(* IEC 61131-3 sources: std_i2980_v2.06_cp053/Source/IMM/ieccontrol/AutoCalibration1 (part 3) *)

(* ---- ABAutoIdentSpeed.pu ---- *)
IMPORT_OVER_LISTFILE
 GET_SYNC_REFTO
, SET_ALARM
, SET_EVENT
, CHECK_REF
, cCompEjector
, cCompMold
, KSYS_Status_OK
, cOptionHydraulic
, tnCalibState_None
, tnCalibState_Running
, tnCalibCommand_Stop
, tnCalibState_Aborted
, cMoveFwd
, cMoveNone
, cMoveBwd
, cMoveDecompAftPlast
, tnCalibState_Error
, cCalibMovements
, nSetup
, tnCalibCommand_None
, tnCalibState_Done
, tnCalibCommand_Start
, tsGlobalIdentSpeedStatus
, tsIdentSpeedMovement
, tnOperationMode
, tyPumpData
, tevRedoIdentSpeedEvent
, tevStopRequest
, tevStartRequest
, tsDeviceId
, tpIdentSpeedMovement
, FBCheckReady
, tevStartRequestData
, tevStopRequestData
, FBIdentSpeedWriteLog
, ABAutoIdentSpeedMeasure
, tnDataState
, KSYS_Status
, tOptionId
, FBTracePendingAlarms
, tevRedoIdentSpeedEventData
, tsVelPre
, tyIdentSpeedMovements
, TON

END_IMPORT

ALGORITHM_BLOCK ABAutoIdentSpeed #DUMMY_EDIT_BLOCK

SYSTEM_VAR
 sv_GlobalIdentMaxSpeedStatus : tsGlobalIdentSpeedStatus;
 sv_EjectorIdentMaxMovement : tsIdentSpeedMovement;
 sv_MoldIdentMaxMovement : tsIdentSpeedMovement;
 sv_InjectionIdentMaxMovement : tsIdentSpeedMovement;
 sv_NozzleIdentMaxMovement : tsIdentSpeedMovement;
 sv_GlobalIdentMinSpeedStatus : tsGlobalIdentSpeedStatus;
 sv_EjectorIdentMinMovement : tsIdentSpeedMovement;
 sv_MoldIdentMinMovement : tsIdentSpeedMovement;
 sv_InjectionIdentMinMovement : tsIdentSpeedMovement;
 sv_NozzleIdentMinMovement : tsIdentSpeedMovement;
 sv_iPendingAlarms : DINT;
 sv_OperationMode : tnOperationMode;
 sv_bAutoIdentRunning : BOOL (* auto calibration active *);
 sv_bCoresActive : BOOL;
 sv_PumpData : tyPumpData;
 sv_DataState : tnDataState;
END_VAR

SYSTEM_OBJECT
 TaskMid : TASK;
 TaskSlow : TASK;
 TaskInject : TASK;
 TaskAnalog : TASK;
 PU_Task_7 : TASK;
 EV_Task_7 : TASK;
 erCalibrationSpeedStopped : ALARM;
 erSetupModeRequiredForCalib : ALARM;
 erCalibCoresActive : ALARM;
 evRedoIdentMaxSpeedStart : tevRedoIdentSpeedEvent;
 evRedoIdentMinSpeedStart : tevRedoIdentSpeedEvent;
 evStopRequest : tevStopRequest;
 evStartRequest : tevStartRequest;
 PU_Task_13 : TASK;
END_OBJECT

VAR
 DeviceIdEjector : tsDeviceId := (CompId:=cCompEjector,IndexId:=1);
 DeviceIdMold : tsDeviceId := (CompId:=cCompMold,IndexId:=1);
 mActMovement : tpIdentSpeedMovement;
 mCalibCounter : DINT;
 mbUseSingleMovement : BOOL;
 fbCheckReady : FBCheckReady;
 evStartRequestData : tevStartRequestData;
 evStopRequestData : tevStopRequestData;
 fbIdentWriteLog : FBIdentSpeedWriteLog;
 miFileCounter : UDINT;
 mbDeleteFiles : BOOL;
 mbLogFileSaved : BOOL := TRUE;
 msFileName : STRING(255);
 mbRestartMeas : BOOL;
 abSpeedMeasure : ABAutoIdentSpeedMeasure;
 mrRefVelocity : REAL;
 mrRefPressure : REAL;
 mrMaxLimitPosition : REAL;
 mrMinLimitPosition : REAL;
 dummy : DINT;
 mrMinPositionFactor : REAL := 0.2 (* 20% of stroke *);
 mrMaxPositionFactor : REAL := 0.8 (* 80% of stroke *);
 mrMaxVelocity : REAL;
 mrMaxPressure : REAL;
 mbVelocityLimitReached : BOOL;
 mbPressureLimitReached : BOOL;
 miErrorNo : INT;
 cIdentSpeedMaxSequence : INT := 100;
 cIdentSpeedMinSequence : INT := 200;
 cIdentSpeedMaxFwdIdent : INT := 101;
 cIdentSpeedMinFwdIdent : INT := 201;
 cIdentSpeedMaxBwdIdent : INT := 102;
 cIdentSpeedMinBwdIdent : INT := 202;
 cIdentSpeedMaxBwdInit : INT := 103;
 cIdentSpeedMinBwdInit : INT := 203;
 cIdentSpeedMaxFwdInit : INT := 104;
 cIdentSpeedMinFwdInit : INT := 204;
 cIdentSpeedMaxFwdStart : INT := 105;
 cIdentSpeedMinFwdStart : INT := 205;
 cIdentSpeedMaxBwdStart : INT := 106;
 cIdentSpeedMinBwdStart : INT := 206;
 cIdentSpeedMaxEnd : INT := 107;
 cIdentSpeedMinEnd : INT := 207;
 mrBwdStopPosition : REAL := 0.05;
 mprActPressure : REFTO REAL;
 mbprActPressureLinked : BOOL;
END_VAR

PROCESS_ALGORITHM paInit ON TaskMid AUTOSTART

VAR_TEMP
 j : DINT;
 k : DINT;
END_VAR

VAR
 i : DINT;
 Status : KSYS_Status;
 rpPosition : REFTO REAL;
 tmpM : tpIdentSpeedMovement;
 pOption : REFTO tOptionId;
END_VAR
#BEGIN_EDIT_BLOCK
(**************************************** WARNING ********************************************
 *** The KEBA Kemro K2 System including software is not intended for safety control tasks! ***
 ***                       For further information see Comment tab!                        ***
 *********************************************************************************************)

i := 1;

rpPosition := GET_SYNC_REFTO('Ejector1.ai_Position', T#0s, Status);
IF Status = KSYS_Status_OK THEN
    sv_GlobalIdentMaxSpeedStatus.pMovements[i] := @sv_EjectorIdentMaxMovement;
    sv_GlobalIdentMinSpeedStatus.pMovements[i] := @sv_EjectorIdentMinMovement;
    i := i + 1;
END_IF;

sv_GlobalIdentMaxSpeedStatus.pMovements[i] := @sv_MoldIdentMaxMovement;
sv_GlobalIdentMinSpeedStatus.pMovements[i] := @sv_MoldIdentMinMovement;
i := i + 1;

pOption := GET_SYNC_REFTO('Nozzle1.sv_Options', T#0s, Status);
IF (Status = KSYS_Status_OK) AND ((pOption^ AND cOptionHydraulic) = cOptionHydraulic) THEN;
    //hydraulic nozzle -> check if ai_Position is available
    rpPosition := GET_SYNC_REFTO('Nozzle1.ai_Position', T#0s, Status);
    IF Status = KSYS_Status_OK THEN
        sv_GlobalIdentMaxSpeedStatus.pMovements[i] := @sv_NozzleIdentMaxMovement;
        sv_GlobalIdentMinSpeedStatus.pMovements[i] := @sv_NozzleIdentMinMovement;
        i := i + 1;
    END_IF;
END_IF;

sv_GlobalIdentMaxSpeedStatus.pMovements[i] := @sv_InjectionIdentMaxMovement;
sv_GlobalIdentMinSpeedStatus.pMovements[i] := @sv_InjectionIdentMinMovement;
i := i + 1;

(* sort them by iOrder *)
FOR k := 1 TO i - 2 DO
    FOR j := 1 TO i - 1 - k DO
        IF sv_GlobalIdentMaxSpeedStatus.pMovements[j]^.iOrder > sv_GlobalIdentMaxSpeedStatus.pMovements[j + 1]^.iOrder THEN
            tmpM := sv_GlobalIdentMaxSpeedStatus.pMovements[j];
            sv_GlobalIdentMaxSpeedStatus.pMovements[j] := sv_GlobalIdentMaxSpeedStatus.pMovements[j + 1];
            sv_GlobalIdentMaxSpeedStatus.pMovements[j + 1] := tmpM;
            tmpM := sv_GlobalIdentMinSpeedStatus.pMovements[j];
            sv_GlobalIdentMinSpeedStatus.pMovements[j] := sv_GlobalIdentMinSpeedStatus.pMovements[j + 1];
            sv_GlobalIdentMinSpeedStatus.pMovements[j + 1] := tmpM;
        END_IF;
    END_FOR;
END_FOR;

sv_GlobalIdentMaxSpeedStatus.iMaxStep := i - 1;
sv_GlobalIdentMinSpeedStatus.iMaxStep := i - 1;

sv_GlobalIdentMaxSpeedStatus.iCurrentStep := 0;
sv_GlobalIdentMaxSpeedStatus.Status := tnCalibState_None;
sv_GlobalIdentMaxSpeedStatus.bInitDone := TRUE;

sv_GlobalIdentMinSpeedStatus.iCurrentStep := 0;
sv_GlobalIdentMinSpeedStatus.Status := tnCalibState_None;
sv_GlobalIdentMinSpeedStatus.bInitDone := TRUE;

STOP_PROCESS_ALGORITHM();

;#END_EDIT_BLOCK END_ALGORITHM

POSTUPDATE_ALGORITHM pAlarmPending ON PU_Task_7 WITH sv_iPendingAlarms

VAR
 fbTracePendingAlarms : FBTracePendingAlarms;
END_VAR
#BEGIN_EDIT_BLOCK
IF ((sv_GlobalIdentMaxSpeedStatus.Status = tnCalibState_Running) OR (sv_GlobalIdentMinSpeedStatus.Status = tnCalibState_Running)) AND
    (sv_iPendingAlarms <> 0) THEN

   dummy := Print('auto max. speed identification stopped because alarms of class 1/2/3 pending');

   //trace all pending alarms
   fbTracePendingAlarms();

   IF (sv_GlobalIdentMaxSpeedStatus.Status = tnCalibState_Running) THEN
      sv_GlobalIdentMaxSpeedStatus.Command := tnCalibCommand_Stop;
      sv_GlobalIdentMaxSpeedStatus.Status := tnCalibState_Aborted;
   ELSE
      sv_GlobalIdentMinSpeedStatus.Command := tnCalibCommand_Stop;
      sv_GlobalIdentMinSpeedStatus.Status := tnCalibState_Aborted;
   END_IF;

   SET_ALARM(Name := erCalibrationSpeedStopped,
             Param1 := miErrorNo);
END_IF;

;#END_EDIT_BLOCK END_ALGORITHM

ALGORITHM aMeasure

VAR
 rActPressure : REAL;
END_VAR
#BEGIN_EDIT_BLOCK
IF mbprActPressureLinked THEN
   rActPressure := mprActPressure^;
ELSE
   rActPressure := 0.0;
END_IF;
abSpeedMeasure.aMeasure(bRestart := mbRestartMeas,
                        rPosition := mActMovement^.prPosition^,
                        rRefVelocity := mrRefVelocity,
                        rActVelocity := mActMovement^.prActVelocity^,
                        rRefPressure := mrRefPressure,
                        rActPressure := rActPressure,
                        rMaxLimitPosition := mrMaxLimitPosition,
                        rMinLimitPosition := mrMinLimitPosition);
mbRestartMeas := FALSE;

;#END_EDIT_BLOCK END_ALGORITHM

PROCESS_ALGORITHM paMeasureFast ON TaskInject

#BEGIN_EDIT_BLOCK
aMeasure();

;#END_EDIT_BLOCK END_ALGORITHM

PROCESS_ALGORITHM paMeasureMid ON TaskAnalog

#BEGIN_EDIT_BLOCK
aMeasure();

;#END_EDIT_BLOCK END_ALGORITHM

ALGORITHM aStartMeasurement

#BEGIN_EDIT_BLOCK
mbRestartMeas := TRUE;
abSpeedMeasure.aReset();
abSpeedMeasure.aMeasure(bRestart := TRUE);
START_PROCESS_ALGORITHM(paMeasureMid);

;#END_EDIT_BLOCK END_ALGORITHM

ALGORITHM aStopMeasurement

#BEGIN_EDIT_BLOCK
STOP_PROCESS_ALGORITHM(paMeasureMid);
abSpeedMeasure.aCloseMeasure();

;#END_EDIT_BLOCK END_ALGORITHM

ALGORITHM aWriteLog

VAR_INPUT
 sFileName : STRING(255) (* file name movement *);
 iFileCounter : UDINT (* actual ident cycle index *);
 bDeleteFiles : BOOL (* delete old files *);
END_VAR
#BEGIN_EDIT_BLOCK
mbLogFileSaved := FALSE;
msFileName := sFileName;
miFileCounter := iFileCounter;
mbDeleteFiles := bDeleteFiles;

START_PROCESS_ALGORITHM(paWriteLog);

;#END_EDIT_BLOCK END_ALGORITHM

PROCESS_ALGORITHM paWriteLog ON TaskSlow

#BEGIN_EDIT_BLOCK
fbIdentWriteLog(sFileName    := msFileName,
                iFileCounter := miFileCounter,
                bDeleteFiles := mbDeleteFiles,
                rMaxVelocity := mrMaxVelocity,
                rMaxPressure := mrMaxPressure,
                bVelocityLimitReached := mbVelocityLimitReached,
                bPressureLimitReached := mbPressureLimitReached);
IF fbIdentWriteLog.bDone THEN
   mbLogFileSaved := TRUE;
ELSE
   mbLogFileSaved := FALSE;
END_IF;
STOP_PROCESS_ALGORITHM();

;#END_EDIT_BLOCK END_ALGORITHM

ALGORITHM aStartMovementFwd

#BEGIN_EDIT_BLOCK
IF mActMovement^.bPositionIncreasingFwd THEN
   mActMovement^.prIdentPosition^ := mActMovement^.prStroke^ * mrMaxPositionFactor;
ELSE
   mActMovement^.prIdentPosition^ := mActMovement^.prStroke^ * mrMinPositionFactor;
END_IF;
mActMovement^.pbMoveIdent^ := TRUE;

evStartRequestData.DeviceId := mActMovement^.DeviceId;
evStartRequestData.MoveDir := cMoveFwd;
IF mActMovement^.MoveId > cMoveNone THEN
   evStartRequestData.MoveId := mActMovement^.MoveId;
ELSE
   evStartRequestData.MoveId := cMoveFwd;
END_IF;

SET_EVENT(evStartRequest, evStartRequestData);

;#END_EDIT_BLOCK END_ALGORITHM

ALGORITHM aStartMovementBwd

#BEGIN_EDIT_BLOCK
IF mActMovement^.bPositionIncreasingFwd THEN
   mActMovement^.prIdentPosition^ := mActMovement^.prStroke^ * mrMinPositionFactor;
ELSE
   mActMovement^.prIdentPosition^ := mActMovement^.prStroke^ * mrMaxPositionFactor;
END_IF;
mActMovement^.pbMoveIdent^ := TRUE;

evStartRequestData.DeviceId := mActMovement^.DeviceId;
evStartRequestData.MoveDir := cMoveBwd;
IF mActMovement^.MoveId > cMoveNone THEN
   evStartRequestData.MoveId := cMoveDecompAftPlast;
ELSE
   evStartRequestData.MoveId := cMoveBwd;
END_IF;

SET_EVENT(evStartRequest, evStartRequestData);

;#END_EDIT_BLOCK END_ALGORITHM

ALGORITHM aStopMovementFwd

#BEGIN_EDIT_BLOCK
evStopRequestData.DeviceId := mActMovement^.DeviceId;
evStopRequestData.MoveDir := cMoveFwd;
evStopRequestData.MoveId := cMoveFwd;
SET_EVENT(evStopRequest, evStopRequestData);
mActMovement^.pbMoveIdent^ := FALSE;
mActMovement^.prIdentPosition^ := 0.0;
mActMovement^.prStopRamp^ := 0.0;

;#END_EDIT_BLOCK END_ALGORITHM

ALGORITHM aStopMovementBwd

#BEGIN_EDIT_BLOCK
evStopRequestData.DeviceId := mActMovement^.DeviceId;
evStopRequestData.MoveDir := cMoveBwd;
IF mActMovement^.MoveId > cMoveNone THEN
   evStopRequestData.MoveId := cMoveDecompAftPlast;
ELSE
   evStopRequestData.MoveId := cMoveBwd;
END_IF;
SET_EVENT(evStopRequest, evStopRequestData);
mActMovement^.pbMoveIdent^ := FALSE;
mActMovement^.prIdentPosition^ := 0.0;
mActMovement^.prStopRamp^ := 0.0;

;#END_EDIT_BLOCK END_ALGORITHM

ALGORITHM aStopMovementError

VAR_INPUT
 sMovementName : STRING(255) (* Movement information *);
END_VAR
#BEGIN_EDIT_BLOCK
sv_GlobalIdentMinSpeedStatus.Status := tnCalibState_Aborted;
mActMovement^.Status := tnCalibState_Error;

dummy := Print('Calib movement "%s" aborted.', sMovementName);

;#END_EDIT_BLOCK END_ALGORITHM

ALGORITHM aCalcMaxSpeedOutput

VAR_INPUT
 rMaxSpeedLimit : REAL (* Maximum speed limit of actual device *);
 rActSpeedLimit : REAL (* Actual speed limit of actual device *);
 rActMaxSpeed : REAL (* Maximum measured speed *);
 bPresLimitReached : BOOL (* Pressure limit reached during movement *);
 bUsePressureMode : BOOL (* Use pressure to check maimum speed limit reached. Otherwise use actual  velocity *);
END_VAR

VAR_OUTPUT
 bMaxDetected : BOOL (* Speed limit detected *);
 rRefSpeed : REAL (* Speed limit for next try *);
 rMaxSpeed : REAL (* Identified max speed *);
END_VAR

VAR
 rSpeedReachedFactor : REAL := 0.95;
 rMaxActSpeed : REAL;
 rMinActSpeed : REAL := 0.0;
 rMinSpeedDifference : REAL := 0.05;
END_VAR
#BEGIN_EDIT_BLOCK
IF (bUsePressureMode) THEN
   IF (rMaxActSpeed = 0.0) THEN
      rMaxActSpeed := rMaxSpeedLimit;
   END_IF;
   IF (bPresLimitReached) THEN
      // reduce refernce value
      rMaxActSpeed := rActSpeedLimit;
      IF (ABS(rMaxActSpeed - rMinActSpeed) < rMinSpeedDifference * rMaxSpeedLimit) THEN
         bMaxDetected := TRUE;
         rMaxSpeed := rMinActSpeed;
         rMinActSpeed := 0.0;
         rMaxActSpeed := 0.0;
      ELSE
         bMaxDetected := FALSE;
         rRefSpeed := 0.5 * (rMaxActSpeed + rMinActSpeed);
      END_IF;
   ELSE
      // ccompare with old value
      IF (rActSpeedLimit = rMaxSpeedLimit) THEN // maximum used at start
         // maximum with tolerance reached
         bMaxDetected := TRUE;
         rMaxSpeed := rMaxSpeedLimit;
         rMinActSpeed := 0.0;
         rMaxActSpeed := 0.0;
      ELSE
         // increase
         rMinActSpeed := rActSpeedLimit;
         IF (ABS(rMaxActSpeed - rMinActSpeed) < rMinSpeedDifference * rMaxSpeedLimit) THEN
            bMaxDetected := TRUE;
            rMaxSpeed := rMinActSpeed;
            rMinActSpeed := 0.0;
            rMaxActSpeed := 0.0;
         ELSE
            rRefSpeed := 0.5 * (rMaxActSpeed + rMinActSpeed);
         END_IF;
      END_IF;
   END_IF;
ELSE
   IF (rActSpeedLimit = rMaxSpeedLimit) THEN // maximum used at start
      IF (rActMaxSpeed > rSpeedReachedFactor * rActSpeedLimit)  THEN
      // maximum with tolerance reached
         bMaxDetected := TRUE;
         rMaxSpeed := rMaxSpeedLimit;
      ELSE
      // actual speed lower than maximum with tolerance
         bMaxDetected := FALSE;
         rRefSpeed := rActMaxSpeed;
         rMaxActSpeed := rActMaxSpeed;
      END_IF;
   ELSE
      IF (rActMaxSpeed > rSpeedReachedFactor * rActSpeedLimit) THEN
      // reference speed with tolerance reached
         bMaxDetected := TRUE;
         rMaxSpeed := rRefSpeed;
      ELSE
      // actual speed lower than reference speed with tolerance reached
      // check calibration of pump/valve
         bMaxDetected := TRUE;
         rMaxSpeed := rRefSpeed;
      END_IF;
   END_IF;
END_IF;

;#END_EDIT_BLOCK END_ALGORITHM

EVENT_ALGORITHM evaRedoMaxEvent ON EV_Task_7 WITH evRedoIdentMaxSpeedStart

VAR_INPUT
 evRedoIdentEventData : tevRedoIdentSpeedEventData (* Event data to start max speed identification *);
END_VAR
#BEGIN_EDIT_BLOCK

START_PROCESS_ALGORITHM(paRedoMax);

;#END_EDIT_BLOCK END_ALGORITHM

PROCESS_ALGORITHM paRedoMax ON TaskMid

VAR_TEMP
 i : DINT;
 bIdentActive : BOOL;
END_VAR
#BEGIN_EDIT_BLOCK
bIdentActive := FALSE;
FOR i:= 1 TO cCalibMovements DO
   IF CHECK_REF(sv_GlobalIdentMaxSpeedStatus.pMovements[i]^) THEN
      IF sv_GlobalIdentMaxSpeedStatus.pMovements[i]^.bRedo THEN
         mActMovement := sv_GlobalIdentMaxSpeedStatus.pMovements[i];
         bIdentActive := TRUE;
         sv_GlobalIdentMaxSpeedStatus.iCurrentStep :=  i;
         mCalibCounter := i;
         IF sv_OperationMode = nSetup THEN
            mbUseSingleMovement := TRUE;
            START_PROCESS_ALGORITHM(paMaxSingleMovement);
         ELSE
            sv_GlobalIdentMaxSpeedStatus.pMovements[i]^.bRedo := FALSE;
            SET_ALARM(erSetupModeRequiredForCalib);
         END_IF;
         EXIT;
      END_IF;
   END_IF;
END_FOR;
IF ((NOT bIdentActive) AND (sv_GlobalIdentMaxSpeedStatus.Status = tnCalibState_Running)) THEN
   sv_GlobalIdentMaxSpeedStatus.Status := tnCalibState_Aborted;
END_IF;

STOP_PROCESS_ALGORITHM();

;#END_EDIT_BLOCK END_ALGORITHM

PROCESS_ALGORITHM paMaxSingleMovement ON TaskMid

VAR
 bMoveBwdDone : BOOL := FALSE;
 bMoveFwdDone : BOOL := FALSE;
 bMoveIdentDone : BOOL := FALSE;
 sFileName : STRING(255);
 iFileCounter : UDINT := 1;
 ConstVis : tsVelPre (* const output for ejector forward movement *);
 ConstVisFwd : tsVelPre (* const output for ejector forward movement *);
 ConstVisBwd : tsVelPre (* const output for ejector forward movement *);
 bMaxFwdRetry : BOOL;
 bMaxBwdRetry : BOOL;
 bMaxFwdDetected : BOOL;
 bMaxBwdDetected : BOOL;
 sMoveName : STRING(32);
 rMaxPressureLimit : REAL;
 rRefSpeedLimit : REAL;
 rSpeedLimitFwd : REAL;
 rSpeedLimitBwd : REAL;
 rMaxRefPressureLimit : REAL;
 sWriteSpeedLimit : STRING(255);
 rVelocitSizeFactor : REAL := 1.0;
 rStartFactor : REAL := 0.1;
 rMinStopRamp : REAL := 1.0;
 rMinStrokeFactor : REAL := 0.5;
 bDelayTimeOffFwdLinked : BOOL;
 bDelayTimeOffBwdLinked : BOOL;
 dDelayTimeOffFwd : TIME;
 dDelayTimeOffBwd : TIME;
 dMinDelayTimeOff : TIME := T#25ms;
END_VAR

(* IecGraph-Code *)

(* init step *)
INITIAL_STEP S_INIT:
Action3 (P);
END_STEP

ACTION Action3: #BEGIN_EDIT_BLOCK
miErrorNo := 0;

ConstVisFwd := mActMovement^.pConstFwdVis^;
ConstVisBwd := mActMovement^.pConstBwdVis^;

sv_GlobalIdentMaxSpeedStatus.Status := tnCalibState_Running;
mActMovement^.Status := tnCalibState_Running;
sMoveName := mActMovement^.sName;

abSpeedMeasure.aInit();

bMaxFwdRetry := FALSE;
bMaxBwdRetry := FALSE;

IF (mActMovement^.rMaxPositionLimitFactor > mActMovement^.rMinPositionLimitFactor) AND
   (mActMovement^.rMinPositionLimitFactor > 0.0) AND (mActMovement^.rMaxPositionLimitFactor < 1.0) THEN
   mrMaxPositionFactor := mActMovement^.rMaxPositionLimitFactor;
   mrMinPositionFactor := mActMovement^.rMinPositionLimitFactor;
ELSE // use deafult values
   mrMaxPositionFactor := 0.8;
   mrMinPositionFactor := 0.2;
END_IF;

mprActPressure := sv_PumpData[mActMovement^.DeviceId.IndexId].prActSysPressure;
IF CHECK_REF(mprActPressure^) THEN
   mbprActPressureLinked := TRUE;
ELSE
   mbprActPressureLinked := FALSE;
END_IF;

IF CHECK_REF(mActMovement^.pdDelayTimeOffFwd^) THEN
   bDelayTimeOffFwdLinked := TRUE;
   dDelayTimeOffFwd := mActMovement^.pdDelayTimeOffFwd^;
ELSE
   bDelayTimeOffFwdLinked := FALSE;
END_IF;
IF CHECK_REF(mActMovement^.pdDelayTimeOffBwd^) THEN
   bDelayTimeOffBwdLinked := TRUE;
   dDelayTimeOffBwd := mActMovement^.pdDelayTimeOffBwd^;
ELSE
   bDelayTimeOffBwdLinked := FALSE;
END_IF;

;#END_EDIT_BLOCK END_ACTION (*Action3*)

(* steps *)
STEP S_RESET:
END_STEP

STEP S_STOP:
AStopSelf (P);
END_STEP

ACTION AStopSelf: #BEGIN_EDIT_BLOCK
sv_GlobalIdentMaxSpeedStatus.Command := tnCalibCommand_None;
sv_bAutoIdentRunning := FALSE;
mActMovement^.bRedo := FALSE;
mActMovement^.prStopRamp^ := 0.0;
mActMovement^.pConstFwdVis^ := ConstVisFwd;
mActMovement^.pConstBwdVis^ := ConstVisBwd;

//release memory
abSpeedMeasure.aEnd();

STOP_PROCESS_ALGORITHM();

;#END_EDIT_BLOCK END_ACTION (*AStopSelf*)
STEP S_MoveStartBwd:
AMoveStartBwd (P);
ACheckMoveStartBwdReady (N);
AMoveStartBwdReady (P0);
END_STEP

ACTION AMoveStartBwd: #BEGIN_EDIT_BLOCK
bMoveBwdDone := FALSE;
miErrorNo := cIdentSpeedMaxBwdInit;
aStartMovementBwd();

;#END_EDIT_BLOCK END_ACTION (*AMoveStartBwd*)
ACTION ACheckMoveStartBwdReady: #BEGIN_EDIT_BLOCK
fbCheckReady(DeviceId := evStartRequestData.DeviceId);
IF fbCheckReady.bReady THEN
   bMoveBwdDone := TRUE;
END_IF;

;#END_EDIT_BLOCK END_ACTION (*ACheckMoveStartBwdReady*)
ACTION AMoveStartBwdReady: #BEGIN_EDIT_BLOCK
aStopMovementBwd();

;#END_EDIT_BLOCK END_ACTION (*AMoveStartBwdReady*)
STEP S_StopMoveStartBwd:
AStopMoveStartBwd (P);
END_STEP

ACTION AStopMoveStartBwd: #BEGIN_EDIT_BLOCK
aStopMovementError(sMovementName := CONCAT(sMoveName, ' max ident Fwd: Bwd to initial position'));

;#END_EDIT_BLOCK END_ACTION (*AStopMoveStartBwd*)
STEP S_CHECK_ALARMS_INITBWD:
END_STEP

STEP S_INITCALIB_FWD:
aInitIdentFwd (P);
END_STEP

ACTION aInitIdentFwd: #BEGIN_EDIT_BLOCK
iFileCounter := 1;
IF (CHECK_REF(mActMovement^.prSizeFactorFwd^)) THEN
   IF (mActMovement^.prSizeFactorFwd^ > 0.0) THEN
      rVelocitSizeFactor := mActMovement^.prSizeFactorFwd^;
   END_IF;
ELSE
   rVelocitSizeFactor := 1.0;
END_IF;
rRefSpeedLimit := mActMovement^.prVelocityLimitFwd^;
rMaxPressureLimit := mActMovement^.prMaxPressureFwd^;
IF CHECK_REF(mActMovement^.prMaxPressureFwdHydr^) THEN
   rMaxRefPressureLimit := mActMovement^.prMaxPressureFwdHydr^;
ELSE
   rMaxRefPressureLimit := rMaxPressureLimit;
END_IF;

dummy := Print('Calib max speed %s Fwd started', sMoveName);

;#END_EDIT_BLOCK END_ACTION (*aInitIdentFwd*)
STEP S_CALIB_FWD:
ADoCalib (P);
AStartMovementFwd (P);
ACheckActMovementFwdReady (N);
AStopMovementFwd (P0);
END_STEP

ACTION ADoCalib: #BEGIN_EDIT_BLOCK
(* start calibration *)
// save actual settings
ConstVis := mActMovement^.pConstFwdVis^;

mActMovement^.pConstFwdVis^.Velocity.Output.rOutputValue := rRefSpeedLimit * rVelocitSizeFactor;
mActMovement^.pConstFwdVis^.Velocity.rMinOutput := 0.0;
mActMovement^.pConstFwdVis^.Pressure.Output.rOutputValue := MAX(mActMovement^.pConstFwdVis^.Pressure.Output.rOutputValue, rMaxPressureLimit);
mActMovement^.pConstFwdVis^.Pressure.Output.rRamp := MAX(1.0e9,ConstVis.Pressure.Output.rRamp);
IF mActMovement^.bPositionIncreasingFwd THEN
   mActMovement^.prIdentPosition^ := mActMovement^.prStroke^ * mrMaxPositionFactor;
   mrMinLimitPosition := rStartFactor * mActMovement^.prIdentPosition^ + (1.0 - rStartFactor) * mActMovement^.prPosition^;
   IF (mActMovement^.prIdentPosition^ - mActMovement^.prPosition^) > 0.0 THEN
      rMinStopRamp := rMinStrokeFactor * rRefSpeedLimit  * rRefSpeedLimit/ ABS(mActMovement^.prIdentPosition^ - mActMovement^.prPosition^);
   ELSE
      rMinStopRamp := 0.0;
   END_IF;
   mActMovement^.prStopRamp^ := MAX(mActMovement^.pConstFwdVis^.Velocity.Output.rRamp, rMinStopRamp);
   mrMaxLimitPosition := mActMovement^.prIdentPosition^;
ELSE
   mActMovement^.prIdentPosition^ := mActMovement^.prStroke^ * mrMinPositionFactor;
   mrMaxLimitPosition := (1.0 - rStartFactor) * mActMovement^.prPosition^ + rStartFactor * mActMovement^.prIdentPosition^;
   IF (mActMovement^.prPosition^ - mActMovement^.prIdentPosition^) > 0.0 THEN
      rMinStopRamp := rMinStrokeFactor * rRefSpeedLimit * rRefSpeedLimit / ABS(mActMovement^.prIdentPosition^ - mActMovement^.prPosition^);
   ELSE
      rMinStopRamp := 0.0;
   END_IF;
   mActMovement^.prStopRamp^ := MAX(mActMovement^.pConstFwdVis^.Velocity.Output.rRamp, rMinStopRamp);
   mrMinLimitPosition := mActMovement^.prIdentPosition^;
END_IF;
mActMovement^.pbMoveIdent^ := TRUE;
bMoveIdentDone := FALSE;

bMaxFwdDetected := FALSE;

mrRefVelocity := rRefSpeedLimit;
mrRefPressure := rMaxRefPressureLimit;
mbRestartMeas := TRUE;

IF bDelayTimeOffFwdLinked THEN
   mActMovement^.pdDelayTimeOffFwd^ := MAX(mActMovement^.pdDelayTimeOffFwd^, dMinDelayTimeOff);
END_IF;
IF bDelayTimeOffBwdLinked THEN
   mActMovement^.pdDelayTimeOffBwd^ := MAX(mActMovement^.pdDelayTimeOffBwd^, dMinDelayTimeOff);
END_IF;

aStartMeasurement();

sWriteSpeedLimit := REAL_TO_STRING(rRefSpeedLimit);
dummy := Print('Calib max output: act. max speed: %s', sWriteSpeedLimit);
miErrorNo := cIdentSpeedMaxFwdIdent;

;#END_EDIT_BLOCK END_ACTION (*ADoCalib*)
ACTION AStartMovementFwd: #BEGIN_EDIT_BLOCK
evStartRequestData.DeviceId := mActMovement^.DeviceId;
evStartRequestData.MoveDir := cMoveFwd;
IF mActMovement^.MoveId > cMoveNone THEN
   evStartRequestData.MoveId := mActMovement^.MoveId;
ELSE
   evStartRequestData.MoveId := cMoveFwd;
END_IF;
SET_EVENT(evStartRequest, evStartRequestData);

;#END_EDIT_BLOCK END_ACTION (*AStartMovementFwd*)
ACTION ACheckActMovementFwdReady: #BEGIN_EDIT_BLOCK
fbCheckReady(DeviceId := evStartRequestData.DeviceId);
IF fbCheckReady.bReady THEN
   bMoveIdentDone := TRUE;
END_IF;

;#END_EDIT_BLOCK END_ACTION (*ACheckActMovementFwdReady*)
ACTION AStopMovementFwd: #BEGIN_EDIT_BLOCK
aStopMeasurement();
aStopMovementFwd();

mActMovement^.pConstFwdVis^ := ConstVis;
mActMovement^.prStopRamp^ := 0.0;

IF bDelayTimeOffFwdLinked THEN
   mActMovement^.pdDelayTimeOffFwd^ := dDelayTimeOffFwd;
END_IF;
IF bDelayTimeOffBwdLinked THEN
   mActMovement^.pdDelayTimeOffBwd^ := dDelayTimeOffBwd;
END_IF;

;#END_EDIT_BLOCK END_ACTION (*AStopMovementFwd*)
STEP S_StopIdentFwd:
AStopIdentFwd (P);
END_STEP

ACTION AStopIdentFwd: #BEGIN_EDIT_BLOCK
aStopMovementError(sMovementName := CONCAT(sMoveName, ' max ident Fwd'));

;#END_EDIT_BLOCK END_ACTION (*AStopIdentFwd*)
STEP S_CHECK_ALARMS_FWD:
END_STEP

STEP S_WRITE_FWD:
AWriteFwd (P);
END_STEP

ACTION AWriteFwd: #BEGIN_EDIT_BLOCK
abSpeedMeasure.aGetMaxValues(rMaxSpeed => mrMaxVelocity,
                             rMaxPressure => mrMaxPressure,
                             bPressureLimitReached => mbPressureLimitReached,
                             bSpeedLimitReached => mbVelocityLimitReached);
sFileName := CONCAT(sMoveName,"_MAXSPEED_FWD_");
aWriteLog(sFileName := sFileName,
          iFileCounter := iFileCounter,
          bDeleteFiles := TRUE);
iFileCounter := iFileCounter + 1;

;#END_EDIT_BLOCK END_ACTION (*AWriteFwd*)
STEP S_AbortedWriteFwd:
AAbortedWriteFwd (P);
END_STEP

ACTION AAbortedWriteFwd: #BEGIN_EDIT_BLOCK
mActMovement^.Status := tnCalibState_Error;

;#END_EDIT_BLOCK END_ACTION (*AAbortedWriteFwd*)
STEP S_CHECK_MAXSPEED_FWD:
ACheckMaxSpeedFwd (P);
END_STEP

ACTION ACheckMaxSpeedFwd: #BEGIN_EDIT_BLOCK
aCalcMaxSpeedOutput(rMaxSpeedLimit := mActMovement^.prVelocityLimitFwd^,
                    rActSpeedLimit := rRefSpeedLimit,
                    rActMaxSpeed := abSpeedMeasure.aGetMaxValues.rMaxSpeed,
                    bPresLimitReached := abSpeedMeasure.aGetMaxValues.bPressureLimitReached,
                    bUsePressureMode := (mrMaxPressure > 0.0));
bMaxFwdDetected := aCalcMaxSpeedOutput.bMaxDetected;
IF (bMaxFwdDetected) THEN
   rSpeedLimitFwd := rRefSpeedLimit;
   dummy := Print('Calib max output %s Fwd finished: max speed fwd = %f$N', sMoveName, rSpeedLimitFwd);
ELSE
   IF abSpeedMeasure.aGetMaxValues.bPressureLimitReached THEN
      sWriteSpeedLimit := REAL_TO_STRING(rRefSpeedLimit);
      dummy := Print('Calib max output: pressure limit reached with act. max speed %s', sWriteSpeedLimit);
   END_IF;
   bMaxFwdRetry := TRUE;
   rRefSpeedLimit := aCalcMaxSpeedOutput.rRefSpeed;
END_IF;

;#END_EDIT_BLOCK END_ACTION (*ACheckMaxSpeedFwd*)
STEP S_MaxFwdRetry:
AStartMovementFwdBwd (P);
ACheckActMovementFwdBwdReady (N);
AStopMovementFwdBwd (P0);
END_STEP

ACTION AStartMovementFwdBwd: #BEGIN_EDIT_BLOCK
bMoveBwdDone := FALSE;
miErrorNo := cIdentSpeedMaxFwdStart;
aStartMovementBwd();

;#END_EDIT_BLOCK END_ACTION (*AStartMovementFwdBwd*)
ACTION ACheckActMovementFwdBwdReady: #BEGIN_EDIT_BLOCK
fbCheckReady(DeviceId := evStartRequestData.DeviceId);
IF fbCheckReady.bReady THEN
   bMoveBwdDone := TRUE;
END_IF;

;#END_EDIT_BLOCK END_ACTION (*ACheckActMovementFwdBwdReady*)
ACTION AStopMovementFwdBwd: #BEGIN_EDIT_BLOCK
aStopMovementBwd();

;#END_EDIT_BLOCK END_ACTION (*AStopMovementFwdBwd*)
STEP S_StopMoveBwd:
AStopMoveBwd (P);
END_STEP

ACTION AStopMoveBwd: #BEGIN_EDIT_BLOCK
aStopMovementError(sMovementName := CONCAT(sMoveName, ' max ident Fwd: Bwd to start position'));

;#END_EDIT_BLOCK END_ACTION (*AStopMoveBwd*)
STEP S_CHECK_ALARMS_RETRYFWD:
END_STEP

STEP S_InitStartMovementBwdFwd:
AInitStartMovementBwdFwd (P);
ACheckInitMovementBwdFwdReady (N);
AStopInitMovementBwdFwd (P0);
END_STEP

ACTION AInitStartMovementBwdFwd: #BEGIN_EDIT_BLOCK
bMoveFwdDone := FALSE;
miErrorNo := cIdentSpeedMaxFwdInit;
aStartMovementFwd();

;#END_EDIT_BLOCK END_ACTION (*AInitStartMovementBwdFwd*)
ACTION ACheckInitMovementBwdFwdReady: #BEGIN_EDIT_BLOCK
fbCheckReady(DeviceId := evStartRequestData.DeviceId);
IF fbCheckReady.bReady THEN
   bMoveFwdDone := TRUE;
END_IF;

;#END_EDIT_BLOCK END_ACTION (*ACheckInitMovementBwdFwdReady*)
ACTION AStopInitMovementBwdFwd: #BEGIN_EDIT_BLOCK
aStopMovementFwd();

;#END_EDIT_BLOCK END_ACTION (*AStopInitMovementBwdFwd*)
STEP S_StopInitMoveFwd:
AStopInitMoveFwd (P);
END_STEP

ACTION AStopInitMoveFwd: #BEGIN_EDIT_BLOCK
aStopMovementError(sMovementName := CONCAT(sMoveName, ' max ident Bwd: Fwd to initial position'));

;#END_EDIT_BLOCK END_ACTION (*AStopInitMoveFwd*)
STEP S_CHECK_ALARMS_STARTBWD:
END_STEP

STEP S_INITCALIB_BWD:
AInitCalibBwd (P);
END_STEP

ACTION AInitCalibBwd: #BEGIN_EDIT_BLOCK
iFileCounter := 1;
IF (CHECK_REF(mActMovement^.prSizeFactorBwd^)) THEN
   IF (mActMovement^.prSizeFactorBwd^ > 0.0) THEN
      rVelocitSizeFactor := mActMovement^.prSizeFactorBwd^;
   END_IF;
ELSE
   rVelocitSizeFactor := 1.0;
END_IF;
rRefSpeedLimit := mActMovement^.prVelocityLimitBwd^;
rMaxPressureLimit := mActMovement^.prMaxPressureBwd^;
IF CHECK_REF(mActMovement^.prMaxPressureBwdHydr^) THEN
   rMaxRefPressureLimit := mActMovement^.prMaxPressureBwdHydr^;
ELSE
   rMaxRefPressureLimit := mActMovement^.prMaxPressureFwd^;
END_IF;

dummy := Print('Calib max speed %s Bwd started', sMoveName);

;#END_EDIT_BLOCK END_ACTION (*AInitCalibBwd*)
STEP S_CALIB_BWD:
ADoCalibBwd (P);
AStartMovementBwd (P);
ACheckActMovementBwdReady (N);
AStopMovementBwd (P0);
END_STEP

ACTION ADoCalibBwd: #BEGIN_EDIT_BLOCK
ConstVis := mActMovement^.pConstBwdVis^;

mActMovement^.pConstBwdVis^.Velocity.Output.rOutputValue := rRefSpeedLimit * rVelocitSizeFactor;
mActMovement^.pConstBwdVis^.Velocity.rMinOutput := 0.0;
mActMovement^.pConstBwdVis^.Pressure.Output.rOutputValue := MAX(mActMovement^.pConstBwdVis^.Pressure.Output.rOutputValue, rMaxPressureLimit);
mActMovement^.pConstBwdVis^.Pressure.Output.rRamp := MAX(1.0e9,ConstVis.Pressure.Output.rRamp);
IF mActMovement^.bPositionIncreasingFwd THEN
   mActMovement^.prIdentPosition^ := mActMovement^.prStroke^ * mrMinPositionFactor;
   mrMaxLimitPosition := rStartFactor * mActMovement^.prIdentPosition^ + (1.0 - rStartFactor) * mActMovement^.prPosition^;
   rMinStopRamp := rRefSpeedLimit / ABS(mActMovement^.prIdentPosition^ - mActMovement^.prPosition^);
   IF (mActMovement^.prPosition^ - mActMovement^.prIdentPosition^) > 0.0 THEN
      rMinStopRamp := rMinStrokeFactor * rRefSpeedLimit * rRefSpeedLimit / ABS(mActMovement^.prIdentPosition^ - mActMovement^.prPosition^);
   ELSE
      rMinStopRamp := 0.0;
   END_IF;
   mActMovement^.prStopRamp^ := MAX(mActMovement^.pConstBwdVis^.Velocity.Output.rRamp, rMinStopRamp);
   mrMinLimitPosition := mActMovement^.prIdentPosition^;
ELSE
   mActMovement^.prIdentPosition^ := mActMovement^.prStroke^ * mrMaxPositionFactor;
   mrMinLimitPosition := rStartFactor * mActMovement^.prPosition^ + (1.0 - rStartFactor) * mActMovement^.prIdentPosition^;
   IF (mActMovement^.prIdentPosition^ - mActMovement^.prPosition^) > 0.0 THEN
      rMinStopRamp := rMinStrokeFactor * rRefSpeedLimit * rRefSpeedLimit / ABS(mActMovement^.prIdentPosition^ - mActMovement^.prPosition^);
   ELSE
      rMinStopRamp := 0.0;
   END_IF;
   mActMovement^.prStopRamp^ := MAX(mActMovement^.pConstBwdVis^.Velocity.Output.rRamp, rMinStopRamp);
   mrMaxLimitPosition := mActMovement^.prIdentPosition^;
END_IF;
mActMovement^.pbMoveIdent^ := TRUE;

bMoveIdentDone := FALSE;

mrRefVelocity := rRefSpeedLimit;
mrRefPressure := rMaxRefPressureLimit;
mbRestartMeas := TRUE;

IF bDelayTimeOffFwdLinked THEN
   mActMovement^.pdDelayTimeOffFwd^ := MAX(mActMovement^.pdDelayTimeOffFwd^, dMinDelayTimeOff);
END_IF;
IF bDelayTimeOffBwdLinked THEN
   mActMovement^.pdDelayTimeOffBwd^ := MAX(mActMovement^.pdDelayTimeOffBwd^, dMinDelayTimeOff);
END_IF;

aStartMeasurement();

sWriteSpeedLimit := REAL_TO_STRING(rRefSpeedLimit);
dummy := Print('Calib max output: act. max speed: %s', sWriteSpeedLimit);
miErrorNo := cIdentSpeedMaxBwdIdent;

;#END_EDIT_BLOCK END_ACTION (*ADoCalibBwd*)
ACTION AStartMovementBwd: #BEGIN_EDIT_BLOCK
evStartRequestData.DeviceId := mActMovement^.DeviceId;
evStartRequestData.MoveDir := cMoveBwd;
IF mActMovement^.MoveId > cMoveNone THEN
   evStartRequestData.MoveId := cMoveDecompAftPlast;
ELSE
   evStartRequestData.MoveId := cMoveBwd;
END_IF;
SET_EVENT(evStartRequest, evStartRequestData);

;#END_EDIT_BLOCK END_ACTION (*AStartMovementBwd*)
ACTION ACheckActMovementBwdReady: #BEGIN_EDIT_BLOCK
fbCheckReady(DeviceId := evStartRequestData.DeviceId);
IF fbCheckReady.bReady THEN
   bMoveIdentDone := TRUE;
END_IF;

;#END_EDIT_BLOCK END_ACTION (*ACheckActMovementBwdReady*)
ACTION AStopMovementBwd: #BEGIN_EDIT_BLOCK
aStopMeasurement();
aStopMovementBwd();

mActMovement^.pConstBwdVis^ := ConstVis;
mActMovement^.prStopRamp^ := 0.0;

IF bDelayTimeOffFwdLinked THEN
   mActMovement^.pdDelayTimeOffFwd^ := dDelayTimeOffFwd;
END_IF;
IF bDelayTimeOffBwdLinked THEN
   mActMovement^.pdDelayTimeOffBwd^ := dDelayTimeOffBwd;
END_IF;

;#END_EDIT_BLOCK END_ACTION (*AStopMovementBwd*)
STEP S_StopCalibBwd:
AStopCalibBwd (P);
END_STEP

ACTION AStopCalibBwd: #BEGIN_EDIT_BLOCK
aStopMovementError(sMovementName := CONCAT(sMoveName, ' max ident Bwd'));

;#END_EDIT_BLOCK END_ACTION (*AStopCalibBwd*)
STEP S_CHECK_ALARMS_BWD:
END_STEP

STEP S_WRITE_BWD:
AWriteBwd (P);
END_STEP

ACTION AWriteBwd: #BEGIN_EDIT_BLOCK
abSpeedMeasure.aGetMaxValues(rMaxSpeed => mrMaxVelocity,
                             rMaxPressure => mrMaxPressure,
                             bPressureLimitReached => mbPressureLimitReached,
                             bSpeedLimitReached => mbVelocityLimitReached);
sFileName := CONCAT(sMoveName,"_MAXSPEED_BWD_");
aWriteLog(sFileName := sFileName,
          iFileCounter := iFileCounter,
          bDeleteFiles := TRUE);
iFileCounter := iFileCounter + 1;

;#END_EDIT_BLOCK END_ACTION (*AWriteBwd*)
STEP S_CHECK_MAXSPEED_BWD:
ACheckMaxSpeedBwd (P);
END_STEP

ACTION ACheckMaxSpeedBwd: #BEGIN_EDIT_BLOCK
aCalcMaxSpeedOutput(rMaxSpeedLimit := mActMovement^.prVelocityLimitBwd^,
                    rActSpeedLimit := rRefSpeedLimit,
                    rActMaxSpeed := abSpeedMeasure.aGetMaxValues.rMaxSpeed,
                    bPresLimitReached := abSpeedMeasure.aGetMaxValues.bPressureLimitReached,
                    bUsePressureMode := (mrMaxPressure > 0.0));
bMaxBwdDetected := aCalcMaxSpeedOutput.bMaxDetected;
IF (bMaxBwdDetected) THEN
   rSpeedLimitBwd := rRefSpeedLimit;
   dummy := Print('Calib max output %s Bwd finished: max speed bwd = %f$N', sMoveName, rSpeedLimitBwd);
ELSE
   IF abSpeedMeasure.aGetMaxValues.bPressureLimitReached THEN
      sWriteSpeedLimit := REAL_TO_STRING(rRefSpeedLimit);
      dummy := Print('Calib max output: pressure limit reached with act. max speed %s', sWriteSpeedLimit);
   END_IF;
   bMaxBwdRetry := TRUE;
   rRefSpeedLimit := aCalcMaxSpeedOutput.rRefSpeed;
END_IF;

;#END_EDIT_BLOCK END_ACTION (*ACheckMaxSpeedBwd*)
STEP S_MaxBwdRetry:
AStartMovementBwdFwd (P);
ACheckActMovementBwdFwdReady (N);
AStopMovementBwdFwd (P0);
END_STEP

ACTION AStartMovementBwdFwd: #BEGIN_EDIT_BLOCK
bMoveFwdDone := FALSE;
miErrorNo := cIdentSpeedMaxBwdStart;
aStartMovementFwd();

;#END_EDIT_BLOCK END_ACTION (*AStartMovementBwdFwd*)
ACTION ACheckActMovementBwdFwdReady: #BEGIN_EDIT_BLOCK
fbCheckReady(DeviceId := evStartRequestData.DeviceId);
IF fbCheckReady.bReady THEN
   bMoveFwdDone := TRUE;
END_IF;

;#END_EDIT_BLOCK END_ACTION (*ACheckActMovementBwdFwdReady*)
ACTION AStopMovementBwdFwd: #BEGIN_EDIT_BLOCK
aStopMovementFwd();

;#END_EDIT_BLOCK END_ACTION (*AStopMovementBwdFwd*)
STEP S_StopMoveFwd:
AStopMoveFwd (P);
END_STEP

ACTION AStopMoveFwd: #BEGIN_EDIT_BLOCK
aStopMovementError(sMovementName := CONCAT(sMoveName, ' max ident Bwd: Fwd to start position'));

;#END_EDIT_BLOCK END_ACTION (*AStopMoveFwd*)
STEP S_CHECK_ALARMS_RETRYBWD:
END_STEP

STEP S_MoveEndBwd:
AMoveEndBwd (P);
ACheckMoveEndBwdReady (N);
AMoveEndBwdReady (P0);
END_STEP

ACTION AMoveEndBwd: #BEGIN_EDIT_BLOCK
bMoveBwdDone := FALSE;

IF mActMovement^.bPositionIncreasingFwd THEN
   mActMovement^.prIdentPosition^ := mrBwdStopPosition;
ELSE
   mActMovement^.prIdentPosition^ := mActMovement^.prStroke^ - mrBwdStopPosition;
END_IF;
mActMovement^.prStopRamp^ := 1.0e10;
mActMovement^.pConstBwdVis^.Pressure.Output.rRamp := MAX(1.0e20,mActMovement^.pConstBwdVis^.Pressure.Output.rRamp);
mActMovement^.pConstBwdVis^.Pressure.rMinOutput := 0.1 * rMaxPressureLimit;
sv_EjectorIdentMinMovement.pConstBwdVis^.Pressure.Output.rRamp := MAX(1.0e10, sv_EjectorIdentMinMovement.pConstBwdVis^.Pressure.Output.rRamp);
sv_EjectorIdentMinMovement.pConstBwdVis^.Pressure.rMinOutput := 0.1 * sv_EjectorIdentMinMovement.prMaxPressureBwd^;

mActMovement^.pbMoveIdent^ := TRUE;

evStartRequestData.DeviceId := mActMovement^.DeviceId;
evStartRequestData.MoveDir := cMoveBwd;
IF mActMovement^.MoveId > cMoveNone THEN
   evStartRequestData.MoveId := cMoveDecompAftPlast;
ELSE
   evStartRequestData.MoveId := cMoveBwd;
END_IF;
miErrorNo := cIdentSpeedMaxEnd;

SET_EVENT(evStartRequest, evStartRequestData);

;#END_EDIT_BLOCK END_ACTION (*AMoveEndBwd*)
ACTION ACheckMoveEndBwdReady: #BEGIN_EDIT_BLOCK
fbCheckReady(DeviceId := evStartRequestData.DeviceId);
IF fbCheckReady.bReady THEN
   bMoveBwdDone := TRUE;
END_IF;

;#END_EDIT_BLOCK END_ACTION (*ACheckMoveEndBwdReady*)
ACTION AMoveEndBwdReady: #BEGIN_EDIT_BLOCK
aStopMovementBwd();

;#END_EDIT_BLOCK END_ACTION (*AMoveEndBwdReady*)
STEP S_StopMoveEndBwd:
AStopMoveEndBwd (P);
END_STEP

ACTION AStopMoveEndBwd: #BEGIN_EDIT_BLOCK
aStopMovementError(sMovementName := CONCAT(sMoveName, ' max ident Bwd to end position'));

;#END_EDIT_BLOCK END_ACTION (*AStopMoveEndBwd*)
STEP S_Done:
ADone (P);
END_STEP

ACTION ADone: #BEGIN_EDIT_BLOCK
mActMovement^.Status := tnCalibState_Done;
sv_GlobalIdentMaxSpeedStatus.Status := tnCalibState_Done;

mActMovement^.prVelocityFwd^ := rSpeedLimitFwd;
mActMovement^.prVelocityBwd^ := rSpeedLimitBwd;

;#END_EDIT_BLOCK END_ACTION (*ADone*)

(* transitions *)
TRANSITION Trans47 (* Trans47 *) FROM S_RESET TO S_STOP :=  #BEGIN_EDIT_BLOCK
mbLogFileSaved
;#END_EDIT_BLOCK
END_TRANSITION

TRANSITION TRestart (* TRestart *) FROM S_STOP TO S_INIT :=  #BEGIN_EDIT_BLOCK
TRUE
;#END_EDIT_BLOCK
END_TRANSITION

TRANSITION TMoveStartBwd (* TMoveStartBwd *) FROM S_INIT TO S_MoveStartBwd :=  #BEGIN_EDIT_BLOCK
TRUE

;#END_EDIT_BLOCK
END_TRANSITION

TRANSITION TInitBwd (* TInitBwd *) FROM S_MoveStartBwd TO S_CHECK_ALARMS_INITBWD :=  #BEGIN_EDIT_BLOCK
bMoveBwdDone
;#END_EDIT_BLOCK
END_TRANSITION

GO_ON_TRANSITION TStopMoveStartBwd (* TStopMoveStartBwd *) FROM S_MoveStartBwd TO S_StopMoveStartBwd :=  #BEGIN_EDIT_BLOCK
sv_GlobalIdentMaxSpeedStatus.Status = tnCalibState_Aborted OR
sv_GlobalIdentMaxSpeedStatus.Status = tnCalibState_None
OR sv_iPendingAlarms <> 0
OR mActMovement^.bRedo = FALSE
;#END_EDIT_BLOCK
END_TRANSITION

GO_ON_TRANSITION TReset (* TReset *) FROM S_StopMoveStartBwd TO S_RESET :=  #BEGIN_EDIT_BLOCK
TRUE
;#END_EDIT_BLOCK
END_TRANSITION

TRANSITION TStartIdent (* TStartIdent *) FROM S_CHECK_ALARMS_INITBWD TO S_INITCALIB_FWD :=  #BEGIN_EDIT_BLOCK
S_CHECK_ALARMS_INITBWD.T > T#100ms
;#END_EDIT_BLOCK
END_TRANSITION

GO_ON_TRANSITION TStopInitBwd (* TStopInitBwd *) FROM S_CHECK_ALARMS_INITBWD TO S_StopMoveStartBwd :=  #BEGIN_EDIT_BLOCK
sv_iPendingAlarms <> 0
;#END_EDIT_BLOCK
END_TRANSITION

TRANSITION TDelay1 (* TDelay1 *) FROM S_INITCALIB_FWD TO S_CALIB_FWD :=  #BEGIN_EDIT_BLOCK
S_INITCALIB_FWD.T>T#1s
;#END_EDIT_BLOCK
END_TRANSITION

TRANSITION TMoveIdentFwdDone (* TMoveIdentFwdDone *) FROM S_CALIB_FWD TO S_CHECK_ALARMS_FWD :=  #BEGIN_EDIT_BLOCK
bMoveIdentDone
;#END_EDIT_BLOCK
END_TRANSITION

GO_ON_TRANSITION TStopIdentFwd (* TStopIdentFwd *) FROM S_CALIB_FWD TO S_StopIdentFwd :=  #BEGIN_EDIT_BLOCK
sv_GlobalIdentMaxSpeedStatus.Status = tnCalibState_Aborted OR
sv_GlobalIdentMaxSpeedStatus.Status = tnCalibState_None
OR sv_iPendingAlarms <> 0
OR mActMovement^.bRedo = FALSE
;#END_EDIT_BLOCK
END_TRANSITION

GO_ON_TRANSITION TReset1 (* TReset1 *) FROM S_StopIdentFwd TO S_RESET :=  #BEGIN_EDIT_BLOCK
TRUE
;#END_EDIT_BLOCK
END_TRANSITION

TRANSITION TStartWriteFwd (* TStartWriteFwd *) FROM S_CHECK_ALARMS_FWD TO S_WRITE_FWD :=  #BEGIN_EDIT_BLOCK
S_CHECK_ALARMS_FWD.T > T#100ms
;#END_EDIT_BLOCK
END_TRANSITION

GO_ON_TRANSITION TStopIdentFwd2 (* TStopIdentFwd2 *) FROM S_CHECK_ALARMS_FWD TO S_StopIdentFwd :=  #BEGIN_EDIT_BLOCK
sv_iPendingAlarms <> 0
;#END_EDIT_BLOCK
END_TRANSITION

TRANSITION TWriteFwd (* TWriteFwd *) FROM S_WRITE_FWD TO S_CHECK_MAXSPEED_FWD :=  #BEGIN_EDIT_BLOCK
mbLogFileSaved
;#END_EDIT_BLOCK
END_TRANSITION

GO_ON_TRANSITION TAbortedWriteFwd (* TAbortedWriteFwd *) FROM S_WRITE_FWD TO S_AbortedWriteFwd :=  #BEGIN_EDIT_BLOCK
sv_GlobalIdentMaxSpeedStatus.Status = tnCalibState_Aborted
;#END_EDIT_BLOCK
END_TRANSITION

GO_ON_TRANSITION TResetAbortedWriteFwd (* TResetAbortedWriteFwd *) FROM S_AbortedWriteFwd TO S_RESET :=  #BEGIN_EDIT_BLOCK
TRUE
;#END_EDIT_BLOCK
END_TRANSITION

TRANSITION TMaxFwdDetected (* TMaxFwdDetected *) FROM S_CHECK_MAXSPEED_FWD TO S_InitStartMovementBwdFwd :=  #BEGIN_EDIT_BLOCK
bMaxFwdDetected
;#END_EDIT_BLOCK
END_TRANSITION

TRANSITION Trans15 (* Trans15 *) FROM S_CHECK_MAXSPEED_FWD TO S_MaxFwdRetry :=  #BEGIN_EDIT_BLOCK
bMaxFwdRetry
;#END_EDIT_BLOCK
END_TRANSITION

TRANSITION TMoveBwdDone (* TMoveBwdDone *) FROM S_MaxFwdRetry TO S_CHECK_ALARMS_RETRYFWD :=  #BEGIN_EDIT_BLOCK
bMoveBwdDone
;#END_EDIT_BLOCK
END_TRANSITION

GO_ON_TRANSITION TStopMoveBwd (* TStopMoveBwd *) FROM S_MaxFwdRetry TO S_StopMoveBwd :=  #BEGIN_EDIT_BLOCK
sv_GlobalIdentMaxSpeedStatus.Status = tnCalibState_Aborted OR
sv_GlobalIdentMaxSpeedStatus.Status = tnCalibState_None
OR sv_iPendingAlarms <> 0
OR mActMovement^.bRedo = FALSE

;#END_EDIT_BLOCK
END_TRANSITION

TRANSITION TReset2 (* TReset2 *) FROM S_StopMoveBwd TO S_RESET :=  #BEGIN_EDIT_BLOCK
TRUE
;#END_EDIT_BLOCK
END_TRANSITION

TRANSITION TRetryFwd (* TRetryFwd *) FROM S_CHECK_ALARMS_RETRYFWD TO S_CALIB_FWD :=  #BEGIN_EDIT_BLOCK
S_CHECK_ALARMS_RETRYFWD.T > T#1s
;#END_EDIT_BLOCK
END_TRANSITION

GO_ON_TRANSITION TStopIdentFwd4 (* TStopIdentFwd4 *) FROM S_CHECK_ALARMS_RETRYFWD TO S_StopMoveBwd :=  #BEGIN_EDIT_BLOCK
sv_iPendingAlarms <> 0
;#END_EDIT_BLOCK
END_TRANSITION

TRANSITION Trans35 (* Trans35 *) FROM S_InitStartMovementBwdFwd TO S_CHECK_ALARMS_STARTBWD :=  #BEGIN_EDIT_BLOCK
bMoveFwdDone
;#END_EDIT_BLOCK
END_TRANSITION

GO_ON_TRANSITION TStopInitMoveFwd (* TStopInitMoveFwd *) FROM S_InitStartMovementBwdFwd TO S_StopInitMoveFwd :=  #BEGIN_EDIT_BLOCK
sv_GlobalIdentMaxSpeedStatus.Status = tnCalibState_Aborted OR
sv_GlobalIdentMaxSpeedStatus.Status = tnCalibState_None
OR sv_iPendingAlarms <> 0
OR mActMovement^.bRedo = FALSE
;#END_EDIT_BLOCK
END_TRANSITION

TRANSITION TResetInitMoveFwd (* TResetInitMoveFwd *) FROM S_StopInitMoveFwd TO S_RESET :=  #BEGIN_EDIT_BLOCK
TRUE
;#END_EDIT_BLOCK
END_TRANSITION

TRANSITION TStartInitBwd (* TStartInitBwd *) FROM S_CHECK_ALARMS_STARTBWD TO S_INITCALIB_BWD :=  #BEGIN_EDIT_BLOCK
S_CHECK_ALARMS_STARTBWD.T > T#100ms
;#END_EDIT_BLOCK
END_TRANSITION

GO_ON_TRANSITION TStopIdentFwd3 (* TStopIdentFwd3 *) FROM S_CHECK_ALARMS_STARTBWD TO S_StopInitMoveFwd :=  #BEGIN_EDIT_BLOCK
sv_iPendingAlarms <> 0
;#END_EDIT_BLOCK
END_TRANSITION

TRANSITION TInitCalibBwd (* TInitCalibBwd *) FROM S_INITCALIB_BWD TO S_CALIB_BWD :=  #BEGIN_EDIT_BLOCK
S_INITCALIB_BWD.T>T#1s
;#END_EDIT_BLOCK
END_TRANSITION

TRANSITION Trans14 (* Trans14 *) FROM S_CALIB_BWD TO S_CHECK_ALARMS_BWD :=  #BEGIN_EDIT_BLOCK
bMoveIdentDone
;#END_EDIT_BLOCK
END_TRANSITION

GO_ON_TRANSITION TStopCalibBwd (* TStopCalibBwd *) FROM S_CALIB_BWD TO S_StopCalibBwd :=  #BEGIN_EDIT_BLOCK
sv_GlobalIdentMaxSpeedStatus.Status = tnCalibState_Aborted OR
sv_GlobalIdentMaxSpeedStatus.Status = tnCalibState_None
OR sv_iPendingAlarms <> 0
OR mActMovement^.bRedo = FALSE
;#END_EDIT_BLOCK
END_TRANSITION

GO_ON_TRANSITION TResetCalibBwd (* TResetCalibBwd *) FROM S_StopCalibBwd TO S_RESET :=  #BEGIN_EDIT_BLOCK
TRUE
;#END_EDIT_BLOCK
END_TRANSITION

TRANSITION TStartWriteBwd (* TStartWriteBwd *) FROM S_CHECK_ALARMS_BWD TO S_WRITE_BWD :=  #BEGIN_EDIT_BLOCK
S_CHECK_ALARMS_BWD.T > T#100ms
;#END_EDIT_BLOCK
END_TRANSITION

GO_ON_TRANSITION TStopCalibBwd2 (* TStopCalibBwd2 *) FROM S_CHECK_ALARMS_BWD TO S_StopCalibBwd :=  #BEGIN_EDIT_BLOCK
sv_iPendingAlarms <> 0
;#END_EDIT_BLOCK
END_TRANSITION

TRANSITION TWriteBwd (* TWriteBwd *) FROM S_WRITE_BWD TO S_CHECK_MAXSPEED_BWD :=  #BEGIN_EDIT_BLOCK
mbLogFileSaved
;#END_EDIT_BLOCK
END_TRANSITION

TRANSITION TMaxBwdDetected (* TMaxBwdDetected *) FROM S_CHECK_MAXSPEED_BWD TO S_MoveEndBwd :=  #BEGIN_EDIT_BLOCK
bMaxBwdDetected
;#END_EDIT_BLOCK
END_TRANSITION

TRANSITION TMaxBwdRetry (* TMaxBwdRetry *) FROM S_CHECK_MAXSPEED_BWD TO S_MaxBwdRetry :=  #BEGIN_EDIT_BLOCK
bMaxBwdRetry
;#END_EDIT_BLOCK
END_TRANSITION

TRANSITION TMoveFwdDone (* TMoveFwdDone *) FROM S_MaxBwdRetry TO S_CHECK_ALARMS_RETRYBWD :=  #BEGIN_EDIT_BLOCK
bMoveFwdDone
;#END_EDIT_BLOCK
END_TRANSITION

GO_ON_TRANSITION TStopMoveFwd (* TStopMoveFwd *) FROM S_MaxBwdRetry TO S_StopMoveFwd :=  #BEGIN_EDIT_BLOCK
sv_GlobalIdentMaxSpeedStatus.Status = tnCalibState_Aborted OR
sv_GlobalIdentMaxSpeedStatus.Status = tnCalibState_None
OR sv_iPendingAlarms <> 0
OR mActMovement^.bRedo = FALSE

;#END_EDIT_BLOCK
END_TRANSITION

TRANSITION TResetBwd (* TResetBwd *) FROM S_StopMoveFwd TO S_RESET :=  #BEGIN_EDIT_BLOCK
TRUE
;#END_EDIT_BLOCK
END_TRANSITION

TRANSITION TRetryBwd (* TRetryBwd *) FROM S_CHECK_ALARMS_RETRYBWD TO S_CALIB_BWD :=  #BEGIN_EDIT_BLOCK
S_CHECK_ALARMS_RETRYBWD.T > T#1s
;#END_EDIT_BLOCK
END_TRANSITION

GO_ON_TRANSITION TStopIdentBwd4 (* TStopIdentBwd4 *) FROM S_CHECK_ALARMS_RETRYBWD TO S_StopMoveFwd :=  #BEGIN_EDIT_BLOCK
sv_iPendingAlarms <> 0
;#END_EDIT_BLOCK
END_TRANSITION

TRANSITION TMoveEndBwdDone (* TMoveEndBwdDone *) FROM S_MoveEndBwd TO S_Done :=  #BEGIN_EDIT_BLOCK
bMoveBwdDone
;#END_EDIT_BLOCK
END_TRANSITION

GO_ON_TRANSITION TStopMoveEndBwd (* TStopMoveEndBwd *) FROM S_MoveEndBwd TO S_StopMoveEndBwd :=  #BEGIN_EDIT_BLOCK
sv_GlobalIdentMaxSpeedStatus.Status = tnCalibState_Aborted OR
sv_GlobalIdentMaxSpeedStatus.Status = tnCalibState_None
OR sv_iPendingAlarms <> 0
;#END_EDIT_BLOCK
END_TRANSITION

GO_ON_TRANSITION TResetMoveEndBwd (* TResetMoveEndBwd *) FROM S_StopMoveEndBwd TO S_RESET :=  #BEGIN_EDIT_BLOCK
TRUE
;#END_EDIT_BLOCK
END_TRANSITION

TRANSITION TDone (* TDone *) FROM S_Done TO S_RESET :=  #BEGIN_EDIT_BLOCK
TRUE
;#END_EDIT_BLOCK
END_TRANSITION

(* end IecGraph-Code *)
(* sfc-code *)
(* end sfc-code *)

END_ALGORITHM

POSTUPDATE_ALGORITHM pMaxCommandListen ON PU_Task_7 WITH sv_GlobalIdentMaxSpeedStatus.Command,sv_GlobalIdentMaxSpeedStatus.bStart

VAR_TEMP
 i : DINT;
END_VAR
#BEGIN_EDIT_BLOCK
//stop all calibrations
// TEST
IF sv_GlobalIdentMaxSpeedStatus.Command = tnCalibCommand_Stop THEN
    sv_GlobalIdentMaxSpeedStatus.bStart := FALSE;
END_IF;
//
IF sv_GlobalIdentMaxSpeedStatus.Command = tnCalibCommand_Stop OR (NOT sv_GlobalIdentMaxSpeedStatus.bStart) THEN
    FOR i:= 1 TO cCalibMovements DO
        IF CHECK_REF(sv_GlobalIdentMaxSpeedStatus.pMovements[i]^) THEN
            IF sv_GlobalIdentMaxSpeedStatus.pMovements[i]^.Status = tnCalibState_Running OR
               sv_GlobalIdentMaxSpeedStatus.pMovements[i]^.bRedo THEN
                sv_GlobalIdentMaxSpeedStatus.pMovements[i]^.Status := tnCalibState_Aborted;
                sv_GlobalIdentMaxSpeedStatus.pMovements[i]^.bRedo := FALSE;//FIXME: check if needed
                sv_GlobalIdentMaxSpeedStatus.Status := tnCalibState_Aborted;
                EXIT;
            END_IF;
        END_IF;
    END_FOR;
    IF (sv_GlobalIdentMaxSpeedStatus.Command = tnCalibCommand_Stop) THEN
       IF (sv_GlobalIdentMaxSpeedStatus.Status <> tnCalibState_Aborted) THEN
          sv_GlobalIdentMaxSpeedStatus.Status := tnCalibState_None;
       END_IF;

    END_IF;
ELSIF (sv_GlobalIdentMaxSpeedStatus.Command = tnCalibCommand_Start) OR (sv_GlobalIdentMaxSpeedStatus.bStart) THEN
    IF sv_OperationMode = nSetup THEN
        mbUseSingleMovement := FALSE;
        START_PROCESS_ALGORITHM(paMaxCalibSequence);
    ELSE
        sv_GlobalIdentMaxSpeedStatus.bStart := FALSE;
        SET_ALARM(erSetupModeRequiredForCalib);
    END_IF;
END_IF;
sv_GlobalIdentMaxSpeedStatus.Command := tnCalibCommand_None;

;#END_EDIT_BLOCK END_ALGORITHM

(*
Coordinate sequential start of auto calib cycle
starts one auto calib movement after the other
*)

PROCESS_ALGORITHM paMaxCalibSequence ON TaskMid

VAR_TEMP
 j : DINT;
 i : DINT;
END_VAR

VAR
 tmpMovements : tyIdentSpeedMovements;
 iMaxMovements : DINT;
 tmpM : tpIdentSpeedMovement;
 ConstBwdVis : tsVelPre;
END_VAR

(* IecGraph-Code *)

(* init step *)
INITIAL_STEP S_INIT:
ASortCalibs (P);
Action108 (P);
END_STEP

ACTION ASortCalibs: #BEGIN_EDIT_BLOCK
sv_GlobalIdentMaxSpeedStatus.Status := tnCalibState_Running;
miErrorNo := 0;

tmpMovements := sv_GlobalIdentMaxSpeedStatus.pMovements;

(* get number of movements *)
FOR i:= 1 TO cCalibMovements DO
    IF NOT CHECK_REF(tmpMovements[i]^)  THEN
        EXIT;
    END_IF;
END_FOR;
iMaxMovements := i -1;

(* sort them by iOrder *)
FOR i := 1 TO iMaxMovements -1 DO
    FOR j := 1 TO iMaxMovements - 1 - i +1 DO
        IF tmpMovements[j]^.iOrder > tmpMovements[j + 1]^.iOrder THEN
            tmpM := tmpMovements[j];
            tmpMovements[j] := tmpMovements[j + 1];
            tmpMovements[j + 1] := tmpM;
        END_IF;
    END_FOR;
END_FOR;

;#END_EDIT_BLOCK END_ACTION (*ASortCalibs*)
ACTION Action108: #BEGIN_EDIT_BLOCK
mCalibCounter := 0;
sv_GlobalIdentMaxSpeedStatus.iCurrentStep := mCalibCounter;

;#END_EDIT_BLOCK END_ACTION (*Action108*)

(* steps *)
STEP S_RESET:
AReset (P);
AStopMovements (N);
AStopSelf (P);
END_STEP

ACTION AReset: #BEGIN_EDIT_BLOCK
sv_bAutoIdentRunning := FALSE;

;#END_EDIT_BLOCK END_ACTION (*AReset*)
ACTION AStopMovements: #BEGIN_EDIT_BLOCK
(* stop all identification movements *)
FOR i:= 1 TO cCalibMovements DO
    IF CHECK_REF(sv_GlobalIdentMaxSpeedStatus.pMovements[i]^) THEN
        IF sv_GlobalIdentMaxSpeedStatus.pMovements[i]^.Status = tnCalibState_Running OR
           sv_GlobalIdentMaxSpeedStatus.pMovements[i]^.bRedo THEN
            sv_GlobalIdentMaxSpeedStatus.pMovements[i]^.Status := tnCalibState_Aborted;
            sv_GlobalIdentMaxSpeedStatus.pMovements[i]^.bRedo := FALSE;//FIXME: check if needed
            EXIT;
        END_IF;
    END_IF;
END_FOR;

;#END_EDIT_BLOCK END_ACTION (*AStopMovements*)
ACTION AStopSelf: #BEGIN_EDIT_BLOCK
sv_GlobalIdentMaxSpeedStatus.bStart := FALSE;
STOP_PROCESS_ALGORITHM();

;#END_EDIT_BLOCK END_ACTION (*AStopSelf*)
STEP Step74:
AAnyCoreActive (N);
END_STEP

STEP Step19:
ASignalStart (P);
END_STEP

ACTION ASignalStart: #BEGIN_EDIT_BLOCK
sv_bAutoIdentRunning := TRUE;

;#END_EDIT_BLOCK END_ACTION (*ASignalStart*)
STEP S_MoveEjectorBack:
AEjectorBack (P);
Action116 (N);
AResetEjectorBack (P0);
END_STEP

ACTION Action116: #BEGIN_EDIT_BLOCK
fbCheckReady(DeviceId := DeviceIdEjector)

;#END_EDIT_BLOCK END_ACTION (*Action116*)
ACTION AResetEjectorBack: #BEGIN_EDIT_BLOCK
miErrorNo := 0;
sv_EjectorIdentMaxMovement.prIdentPosition^ := 0.0;
sv_EjectorIdentMaxMovement.prStopRamp^ := 0.0;
sv_EjectorIdentMaxMovement.pbMoveIdent^ := FALSE;
sv_EjectorIdentMaxMovement.pConstBwdVis^ := ConstBwdVis;

;#END_EDIT_BLOCK END_ACTION (*AResetEjectorBack*)
STEP S_StopEjector:
AStopEjeMovement (P);
END_STEP

STEP S_MoveMoldBack:
AMoldBack (P);
Action118 (N);
AResetMoldBack (P0);
END_STEP

ACTION Action118: #BEGIN_EDIT_BLOCK
fbCheckReady(DeviceId := DeviceIdMold)

;#END_EDIT_BLOCK END_ACTION (*Action118*)
ACTION AResetMoldBack: #BEGIN_EDIT_BLOCK
miErrorNo := 0;
sv_MoldIdentMaxMovement.prIdentPosition^ := 0.0;
sv_MoldIdentMaxMovement.prStopRamp^ := 0.0;
sv_MoldIdentMaxMovement.pbMoveIdent^ := FALSE;
sv_MoldIdentMaxMovement.pConstBwdVis^ := ConstBwdVis;

;#END_EDIT_BLOCK END_ACTION (*AResetMoldBack*)
STEP S_StopMold:
AStopMoldMovement (P);
END_STEP

STEP S_CALIB_SINGLE:
AStartMovementStart (P);
END_STEP

ACTION AStartMovementStart: #BEGIN_EDIT_BLOCK
IF mCalibCounter < iMaxMovements THEN
   mCalibCounter := mCalibCounter +1;
   tmpMovements[mCalibCounter]^.bRedo := TRUE;
END_IF;

;#END_EDIT_BLOCK END_ACTION (*AStartMovementStart*)
STEP S_CHECKNEXT:
END_STEP

STEP S_StopIdent:
AStopIdent (P);
END_STEP

ACTION AStopIdent: #BEGIN_EDIT_BLOCK
sv_GlobalIdentMaxSpeedStatus.Status := tnCalibState_Done;

;#END_EDIT_BLOCK END_ACTION (*AStopIdent*)

(* transitions *)
TRANSITION Trans50 (* Trans50 *) FROM S_RESET TO S_INIT :=  #BEGIN_EDIT_BLOCK
TRUE
;#END_EDIT_BLOCK
END_TRANSITION

TRANSITION Trans80 (* Trans80 *) FROM S_INIT TO Step19 :=  #BEGIN_EDIT_BLOCK
NOT sv_bCoresActive AND
sv_iPendingAlarms = 0
;#END_EDIT_BLOCK
(*Comment : Start with moving ejector and
mold in backward position, check if any failure
occured.
After that start the calibration cycle, if no alarm is
pending*)
END_TRANSITION

GO_ON_TRANSITION Trans87 (* Trans87 *) FROM S_INIT TO Step74 :=  #BEGIN_EDIT_BLOCK
sv_bCoresActive OR
sv_iPendingAlarms > 0
;#END_EDIT_BLOCK
END_TRANSITION

TRANSITION Trans88 (* Trans88 *) FROM Step74 TO S_RESET :=  #BEGIN_EDIT_BLOCK
TRUE

;#END_EDIT_BLOCK
END_TRANSITION

TRANSITION Trans18 (* Trans18 *) FROM Step19 TO S_MoveEjectorBack :=  #BEGIN_EDIT_BLOCK
TRUE
;#END_EDIT_BLOCK
END_TRANSITION

TRANSITION Trans72 (* Trans72 *) FROM S_MoveEjectorBack TO S_MoveMoldBack :=  #BEGIN_EDIT_BLOCK
fbCheckReady.bReady AND
sv_iPendingAlarms = 0
;#END_EDIT_BLOCK
END_TRANSITION

GO_ON_TRANSITION Trans83 (* Trans83 *) FROM S_MoveEjectorBack TO S_StopEjector :=  #BEGIN_EDIT_BLOCK
sv_GlobalIdentMaxSpeedStatus.Status = tnCalibState_Aborted OR
sv_GlobalIdentMaxSpeedStatus.Status = tnCalibState_None
OR sv_iPendingAlarms <> 0
;#END_EDIT_BLOCK
END_TRANSITION

TRANSITION Trans84 (* Trans84 *) FROM S_StopEjector TO S_RESET :=  #BEGIN_EDIT_BLOCK
TRUE

;#END_EDIT_BLOCK
END_TRANSITION

TRANSITION Trans81 (* Trans81 *) FROM S_MoveMoldBack TO S_CALIB_SINGLE :=  #BEGIN_EDIT_BLOCK
fbCheckReady.bReady AND
sv_iPendingAlarms = 0
;#END_EDIT_BLOCK
END_TRANSITION

GO_ON_TRANSITION Trans85 (* Trans85 *) FROM S_MoveMoldBack TO S_StopMold :=  #BEGIN_EDIT_BLOCK
sv_GlobalIdentMaxSpeedStatus.Status = tnCalibState_Aborted OR
sv_GlobalIdentMaxSpeedStatus.Status = tnCalibState_None
OR sv_iPendingAlarms <> 0
;#END_EDIT_BLOCK
END_TRANSITION

TRANSITION Trans86 (* Trans86 *) FROM S_StopMold TO S_RESET :=  #BEGIN_EDIT_BLOCK
TRUE
;#END_EDIT_BLOCK
END_TRANSITION

TRANSITION TCheckActMoveReady (* TCheckActMoveReady *) FROM S_CALIB_SINGLE TO S_CHECKNEXT :=  #BEGIN_EDIT_BLOCK
tmpMovements[mCalibCounter]^.bRedo = FALSE AND
NOT(sv_GlobalIdentMaxSpeedStatus.Status = tnCalibState_Aborted OR
    sv_GlobalIdentMaxSpeedStatus.Status = tnCalibState_Error)
;#END_EDIT_BLOCK
END_TRANSITION

GO_ON_TRANSITION TCheckError (* TCheckError *) FROM S_CALIB_SINGLE TO S_RESET :=  #BEGIN_EDIT_BLOCK
sv_GlobalIdentMaxSpeedStatus.Status = tnCalibState_Aborted OR
sv_GlobalIdentMaxSpeedStatus.Status = tnCalibState_Error OR
iMaxMovements = 0
;#END_EDIT_BLOCK
END_TRANSITION

TRANSITION TNextUnit (* TNextUnit *) FROM S_CHECKNEXT TO S_CALIB_SINGLE :=  #BEGIN_EDIT_BLOCK
mCalibCounter < iMaxMovements
;#END_EDIT_BLOCK
END_TRANSITION

TRANSITION TStopIdent (* TStopIdent *) FROM S_CHECKNEXT TO S_StopIdent :=  #BEGIN_EDIT_BLOCK
mCalibCounter >= iMaxMovements
;#END_EDIT_BLOCK
END_TRANSITION

TRANSITION TReset (* TReset *) FROM S_StopIdent TO S_RESET :=  #BEGIN_EDIT_BLOCK
TRUE
;#END_EDIT_BLOCK
END_TRANSITION

(* end IecGraph-Code *)
(* sfc-code *)

(* stand alone actions *)
ACTION AEjectorBack: #BEGIN_EDIT_BLOCK
miErrorNo := cIdentSpeedMaxSequence;

IF sv_EjectorIdentMaxMovement.bPositionIncreasingFwd THEN
   sv_EjectorIdentMaxMovement.prIdentPosition^ := mrBwdStopPosition;
ELSE
   sv_EjectorIdentMaxMovement.prIdentPosition^ := sv_EjectorIdentMaxMovement.prStroke^ - mrBwdStopPosition;
END_IF;
sv_EjectorIdentMaxMovement.prStopRamp^ := 1.0e10;
ConstBwdVis := sv_EjectorIdentMaxMovement.pConstBwdVis^;
sv_EjectorIdentMaxMovement.pConstBwdVis^.Pressure.Output.rRamp := MAX(1.0e10, sv_EjectorIdentMaxMovement.pConstBwdVis^.Pressure.Output.rRamp);
sv_EjectorIdentMaxMovement.pConstBwdVis^.Pressure.rMinOutput := 0.1 * sv_EjectorIdentMaxMovement.prMaxPressureBwd^;
sv_EjectorIdentMaxMovement.pbMoveIdent^ := TRUE;

evStartRequestData.DeviceId := DeviceIdEjector;
evStartRequestData.MoveDir := cMoveBwd;
evStartRequestData.MoveId := cMoveBwd;
SET_EVENT(evStartRequest, evStartRequestData);

;#END_EDIT_BLOCK END_ACTION (*AEjectorBack*)
ACTION AMoldBack: #BEGIN_EDIT_BLOCK
miErrorNo := cIdentSpeedMaxSequence;

IF sv_MoldIdentMaxMovement.bPositionIncreasingFwd THEN
   sv_MoldIdentMaxMovement.prIdentPosition^ := mrBwdStopPosition;
ELSE
   sv_MoldIdentMaxMovement.prIdentPosition^ := sv_MoldIdentMaxMovement.prStroke^ - mrBwdStopPosition;
END_IF;
sv_MoldIdentMaxMovement.prStopRamp^ := 1.0e10;
ConstBwdVis := sv_MoldIdentMaxMovement.pConstBwdVis^;
sv_MoldIdentMaxMovement.pConstBwdVis^.Pressure.Output.rRamp := MAX(1.0e10, sv_MoldIdentMaxMovement.pConstBwdVis^.Pressure.Output.rRamp);
sv_MoldIdentMaxMovement.pConstBwdVis^.Pressure.rMinOutput := 0.1 * sv_MoldIdentMaxMovement.prMaxPressureBwd^;
sv_MoldIdentMaxMovement.pbMoveIdent^ := TRUE;

evStartRequestData.DeviceId := DeviceIdMold;
evStartRequestData.MoveDir := cMoveBwd;
evStartRequestData.MoveId := cMoveBwd;
SET_EVENT(evStartRequest, evStartRequestData);

;#END_EDIT_BLOCK END_ACTION (*AMoldBack*)
ACTION AStopEjeMovement: #BEGIN_EDIT_BLOCK
evStopRequestData.DeviceId := DeviceIdEjector;
evStopRequestData.MoveDir := cMoveBwd;
evStopRequestData.MoveId := cMoveBwd;
SET_EVENT(evStopRequest, evStopRequestData);
IF sv_GlobalIdentMaxSpeedStatus.Status <> tnCalibState_None THEN
    sv_GlobalIdentMaxSpeedStatus.Status := tnCalibState_Aborted;
END_IF;

;#END_EDIT_BLOCK END_ACTION (*AStopEjeMovement*)
ACTION AStopMoldMovement: #BEGIN_EDIT_BLOCK
evStopRequestData.DeviceId := DeviceIdMold;
evStopRequestData.MoveDir := cMoveBwd;
evStopRequestData.MoveId := cMoveBwd;
SET_EVENT(evStopRequest, evStopRequestData);
IF sv_GlobalIdentMaxSpeedStatus.Status <> tnCalibState_None THEN
    sv_GlobalIdentMaxSpeedStatus.Status := tnCalibState_Aborted;
END_IF;

;#END_EDIT_BLOCK END_ACTION (*AStopMoldMovement*)
ACTION AAnyCoreActive: #BEGIN_EDIT_BLOCK
IF sv_bCoresActive THEN
   SET_ALARM(erCalibCoresActive);
END_IF;
sv_GlobalIdentMaxSpeedStatus.Status := tnCalibState_Aborted;

;#END_EDIT_BLOCK END_ACTION (*AAnyCoreActive*)

(* exits *)

EXIT_TRANSITION E_NotSetupMode := #BEGIN_EDIT_BLOCK
sv_OperationMode <> nSetup
;#END_EDIT_BLOCK
PRIORITY 1 WITH  INITIAL_STEP S_RESET: END_STEP
END_TRANSITION
(* end sfc-code *)

END_ALGORITHM

ALGORITHM aRound

VAR_INPUT
 rActNumber : REAL;
 rStep : REAL;
END_VAR

VAR_OUTPUT
 rRoundedNumber : REAL;
END_VAR

VAR
 rRealValue : REAL;
END_VAR
#BEGIN_EDIT_BLOCK
IF (rStep > 0.0) THEN
   rRealValue := (0.999 + rActNumber / rStep);
   rRoundedNumber := DINT_TO_REAL(TRUNC_TO_DINT(rRealValue)) * rStep;
ELSE
   rRoundedNumber := rActNumber;
END_IF;

;#END_EDIT_BLOCK END_ALGORITHM

ALGORITHM aCalcMinSpeedOutput

VAR_INPUT
 bStart : BOOL (* Restart calculation of reference for min speed calibration *);
 rMaxSpeedLimit : REAL (* Maximum speed limit of actual device *);
 rActRefSpeed : REAL (* Actual speed limit of actual device *);
 rActMinSpeed : REAL (* Minimum measured speed *);
 bUnstable : BOOL (* Measured speed unstable *);
 bTimeOut : BOOL (* Timeout during movement aof actual device *);
END_VAR

VAR_OUTPUT
 bMinDetected : BOOL (* Speed limit detected *);
 rRefSpeed : REAL (* Speed limit for next try *);
 rMinSpeed : REAL (* Identified min output *);
END_VAR

VAR
 rMaxRefSpeed : REAL;
 rMinRefSpeed : REAL := 0.0;
 rMFactorMaxMinLimit : REAL := 0.2;
END_VAR
#BEGIN_EDIT_BLOCK
IF bStart THEN
   rMaxRefSpeed := rMaxSpeedLimit;
   rMinRefSpeed := 0.0;
END_IF;
IF (bUnstable OR bTimeOut) THEN
   // increase speed
   IF (rActRefSpeed >= rMFactorMaxMinLimit * rMaxSpeedLimit) THEN
      bMinDetected := TRUE;
      rMinSpeed := rActRefSpeed;
      RETURN;
   END_IF;
   rMinRefSpeed := rActRefSpeed;
   bMinDetected := FALSE;
  IF (rMaxRefSpeed - rMinRefSpeed) < (0.0025 * rMaxSpeedLimit) THEN
  // difference to low to maximum - stop or increase maximum?
      bMinDetected := TRUE;
      rMinSpeed := rMaxRefSpeed;
   ELSIF (rMaxRefSpeed < rMaxSpeedLimit) AND (rMinRefSpeed > 0.0) THEN
      rRefSpeed := 0.5 * (rMaxRefSpeed + rMinRefSpeed);
      bMinDetected := FALSE;
   ELSE
      rRefSpeed := rActRefSpeed + 0.01 * rMaxSpeedLimit;
      IF (rRefSpeed >= rMaxSpeedLimit) THEN
         bMinDetected := TRUE;
         rMinSpeed := rMaxSpeedLimit;
      END_IF;
   END_IF;
ELSE
   // reduce speed
   rMaxRefSpeed := rActRefSpeed;
   IF (rMaxRefSpeed - rMinRefSpeed) < (0.0025 * rMaxSpeedLimit) THEN
      bMinDetected := TRUE;
      rMinSpeed := rActRefSpeed;
   ELSE
      bMinDetected := FALSE;
      rRefSpeed := 0.5 * (rMaxRefSpeed + rMinRefSpeed);
   END_IF;
END_IF;

;#END_EDIT_BLOCK END_ALGORITHM

PROCESS_ALGORITHM paRedoMin ON TaskMid

VAR_TEMP
 i : DINT;
 bIdentActive : BOOL;
END_VAR
#BEGIN_EDIT_BLOCK
bIdentActive := FALSE;
FOR i:= 1 TO cCalibMovements DO
   IF CHECK_REF(sv_GlobalIdentMinSpeedStatus.pMovements[i]^) THEN
      IF sv_GlobalIdentMinSpeedStatus.pMovements[i]^.bRedo THEN
         mActMovement := sv_GlobalIdentMinSpeedStatus.pMovements[i];
         bIdentActive := TRUE;
         sv_GlobalIdentMinSpeedStatus.iCurrentStep :=  i;
         mCalibCounter := i;
         IF sv_OperationMode = nSetup THEN
            mbUseSingleMovement := TRUE;
            START_PROCESS_ALGORITHM(paMinSingleMovement);
         ELSE
            sv_GlobalIdentMinSpeedStatus.pMovements[i]^.bRedo := FALSE;
            SET_ALARM(erSetupModeRequiredForCalib);
         END_IF;
         EXIT;
      END_IF;
   END_IF;
END_FOR;
IF ((NOT bIdentActive) AND (sv_GlobalIdentMinSpeedStatus.Status = tnCalibState_Running)) THEN
   sv_GlobalIdentMinSpeedStatus.Status := tnCalibState_Done;
END_IF;

STOP_PROCESS_ALGORITHM();

;#END_EDIT_BLOCK END_ALGORITHM

EVENT_ALGORITHM evaRedoMinEvent ON EV_Task_7 WITH evRedoIdentMinSpeedStart

VAR_INPUT
 evRedoIdentEventData : tevRedoIdentSpeedEventData (* Event data to start min speed identification *);
END_VAR
#BEGIN_EDIT_BLOCK

START_PROCESS_ALGORITHM(paRedoMin);

;#END_EDIT_BLOCK END_ALGORITHM

PROCESS_ALGORITHM paMinSingleMovement ON TaskMid

VAR
 bMoveBwdDone : BOOL := FALSE;
 bMoveFwdDone : BOOL := FALSE;
 bMoveIdentDone : BOOL := FALSE;
 sFileName : STRING(255);
 iFileCounter : UDINT := 1;
 ConstVisFwd : tsVelPre (* const output for ejector forward movement *);
 ConstVisBwd : tsVelPre (* const output for ejector forward movement *);
 bMinFwdRetry : BOOL;
 bMinBwdRetry : BOOL;
 bMinFwdDetected : BOOL;
 bMinBwdDetected : BOOL;
 sMoveName : STRING(32);
 rMaxPressureLimit : REAL := 150.0;
 rRefSpeedLimit : REAL;
 rSpeedLimitFwd : REAL;
 rSpeedLimitBwd : REAL;
 bTimeOut : BOOL;
 bStopUnstable : BOOL;
 dMaxMoveTime : TIME;
 dMaxMoveTimeSaveFwd : TIME;
 dMaxMoveTimeSaveBwd : TIME;
 TimeOut : TON;
 rMoveStrokeTime : REAL;
 rStartFactor : REAL := 0.1;
 rMaxRefPressureLimit : REAL;
 sWriteSpeedLimit : STRING(255);
 dMoveTimeLimit : TIME := T#2m;
 bMoveTimeLimited : BOOL;
 dMoveTimeOffset : TIME := T#5s;
 rStartPosition : REAL;
 rMinMovementPosition : REAL;
 rVelocitSizeFactor : REAL := 1.0;
 rMinStopRamp : REAL := 1.0;
 rMinStrokeFactor : REAL := 2.0;
 rMaxPressureFwd : REAL;
 rMaxPressureBwd : REAL;
 rPressureFactorFwd : REAL;
 rPressureFactorBwd : REAL;
 rPressureStep : REAL := 5.0;
END_VAR

(* IecGraph-Code *)

(* init step *)
INITIAL_STEP S_INIT:
Action3 (P);
END_STEP

ACTION Action3: #BEGIN_EDIT_BLOCK
miErrorNo := 0;

sv_GlobalIdentMinSpeedStatus.Status := tnCalibState_Running;
mActMovement^.Status := tnCalibState_Running;
sMoveName := mActMovement^.sName;

abSpeedMeasure.aInit();

bMinFwdRetry := FALSE;
bMinBwdRetry := FALSE;

dMaxMoveTimeSaveFwd := mActMovement^.pdMaxMoveTimeFwd^;
dMaxMoveTimeSaveBwd := mActMovement^.pdMaxMoveTimeBwd^;

ConstVisFwd := mActMovement^.pConstFwdVis^;
ConstVisBwd := mActMovement^.pConstBwdVis^;

rSpeedLimitFwd := mActMovement^.prVelocityFwd^;
rSpeedLimitBwd := mActMovement^.prVelocityBwd^;

IF (mActMovement^.rMaxPositionLimitFactor > mActMovement^.rMinPositionLimitFactor) AND
   (mActMovement^.rMinPositionLimitFactor > 0.0) AND (mActMovement^.rMaxPositionLimitFactor < 1.0) THEN
   mrMaxPositionFactor := mActMovement^.rMaxPositionLimitFactor;
   mrMinPositionFactor := mActMovement^.rMinPositionLimitFactor;
ELSE // use deafult values
   mrMaxPositionFactor := 0.8;
   mrMinPositionFactor := 0.2;
END_IF;

rMaxPressureFwd := 0.0;
rMaxPressureBwd := 0.0;
mprActPressure := sv_PumpData[mActMovement^.DeviceId.IndexId].prActSysPressure;
IF CHECK_REF(mprActPressure^) THEN
   mbprActPressureLinked := TRUE;
ELSE
   mbprActPressureLinked := FALSE;
END_IF;

;#END_EDIT_BLOCK END_ACTION (*Action3*)

(* steps *)
STEP S_RESET:
END_STEP

STEP S_STOP:
AStopSelf (P);
END_STEP

ACTION AStopSelf: #BEGIN_EDIT_BLOCK
IF (sv_GlobalIdentMinSpeedStatus.Status = tnCalibState_Aborted) THEN
   mActMovement^.prVelocityFwd^ := rSpeedLimitFwd;
   mActMovement^.prVelocityBwd^ := rSpeedLimitBwd;
END_IF;
sv_GlobalIdentMinSpeedStatus.Command := tnCalibCommand_None;
sv_bAutoIdentRunning := FALSE;
mActMovement^.bRedo := FALSE;
mActMovement^.pdMaxMoveTimeFwd^ := dMaxMoveTimeSaveFwd;
mActMovement^.pdMaxMoveTimeBwd^ := dMaxMoveTimeSaveBwd;
mActMovement^.prStopRamp^ := 0.0;
mActMovement^.pConstFwdVis^ := ConstVisFwd;
mActMovement^.pConstBwdVis^ := ConstVisBwd;

//release memory
abSpeedMeasure.aEnd();

STOP_PROCESS_ALGORITHM();

;#END_EDIT_BLOCK END_ACTION (*AStopSelf*)
STEP S_MoveStartBwd:
AMoveStartBwd (P);
ACheckMoveStartBwdReady (N);
AMoveStartBwdReady (P0);
END_STEP

ACTION AMoveStartBwd: #BEGIN_EDIT_BLOCK
bMoveBwdDone := FALSE;
miErrorNo := cIdentSpeedMinBwdInit;
aStartMovementBwd();

;#END_EDIT_BLOCK END_ACTION (*AMoveStartBwd*)
ACTION ACheckMoveStartBwdReady: #BEGIN_EDIT_BLOCK
fbCheckReady(DeviceId := evStartRequestData.DeviceId);
IF fbCheckReady.bReady THEN
   bMoveBwdDone := TRUE;
END_IF;

;#END_EDIT_BLOCK END_ACTION (*ACheckMoveStartBwdReady*)
ACTION AMoveStartBwdReady: #BEGIN_EDIT_BLOCK
aStopMovementBwd();

;#END_EDIT_BLOCK END_ACTION (*AMoveStartBwdReady*)
STEP S_StopMoveStartBwd:
AStopMoveErrorStartBwd (P);
END_STEP

ACTION AStopMoveErrorStartBwd: #BEGIN_EDIT_BLOCK
aStopMovementError(sMovementName := CONCAT(sMoveName, ' min ident Fwd: Bwd to initial position'));

;#END_EDIT_BLOCK END_ACTION (*AStopMoveErrorStartBwd*)
STEP S_CHECK_ALARMS_INITBWD:
END_STEP

STEP S_INITCALIB_FWD:
aInitIdentFwd (P);
END_STEP

ACTION aInitIdentFwd: #BEGIN_EDIT_BLOCK
iFileCounter := 1;
IF (CHECK_REF(mActMovement^.prSizeFactorFwd^)) THEN
   IF (mActMovement^.prSizeFactorFwd^ > 0.0) THEN
      rVelocitSizeFactor := mActMovement^.prSizeFactorFwd^;
   END_IF;
ELSE
   rVelocitSizeFactor := 1.0;
END_IF;
rRefSpeedLimit := 0.01 * mActMovement^.prVelocityLimitFwd^;
rMaxPressureLimit := mActMovement^.prMaxPressureFwd^;
IF CHECK_REF(mActMovement^.prMaxPressureFwdHydr^) THEN
   rMaxRefPressureLimit := mActMovement^.prMaxPressureFwdHydr^;
   IF (rMaxRefPressureLimit > 0.0) THEN
      rPressureFactorFwd := rMaxPressureLimit / rMaxRefPressureLimit;
   ELSE
      rPressureFactorFwd := 1.0;
   END_IF;
ELSE
   rMaxRefPressureLimit := mActMovement^.prMaxPressureFwd^;
   rPressureFactorFwd := 1.0;
END_IF;

aCalcMinSpeedOutput.bStart := TRUE;

dummy := Print('Calib min output %s Fwd started', sMoveName);

;#END_EDIT_BLOCK END_ACTION (*aInitIdentFwd*)
STEP S_CALIB_FWD:
ADoCalib (P);
AStartMovementFwd (P);
ACheckActMovementFwdReady (N);
AStopMovementFwd (P0);
END_STEP

ACTION ADoCalib: #BEGIN_EDIT_BLOCK
// save actual settings
mActMovement^.pConstFwdVis^.Velocity.Output.rOutputValue := rRefSpeedLimit * rVelocitSizeFactor;
mActMovement^.pConstFwdVis^.Velocity.rMinOutput := 0.0;
mActMovement^.pConstFwdVis^.Pressure.Output.rOutputValue := MAX(mActMovement^.pConstFwdVis^.Pressure.Output.rOutputValue, rMaxPressureLimit);
mActMovement^.pConstFwdVis^.Pressure.Output.rRamp := MAX(1.0e10, ConstVisFwd.Pressure.Output.rRamp);
IF mActMovement^.bPositionIncreasingFwd THEN
   mActMovement^.prIdentPosition^ := mActMovement^.prStroke^ * mrMaxPositionFactor;
   mrMinLimitPosition := rStartFactor * mActMovement^.prIdentPosition^ + (1.0 - rStartFactor) * mActMovement^.prPosition^;
   IF (mActMovement^.prIdentPosition^ - mActMovement^.prPosition^) > 0.0 THEN
      rMinStopRamp := rMinStrokeFactor * rRefSpeedLimit  * rRefSpeedLimit / ABS(mActMovement^.prIdentPosition^ - mActMovement^.prPosition^);
   ELSE
      rMinStopRamp := 0.0;
   END_IF;
   mActMovement^.prStopRamp^ := MAX(mActMovement^.pConstFwdVis^.Velocity.Output.rRamp, rMinStopRamp);
   mrMaxLimitPosition := mActMovement^.prIdentPosition^ - 0.5 * rRefSpeedLimit  * rRefSpeedLimit / mActMovement^.prStopRamp^;
ELSE
   mActMovement^.prIdentPosition^ := mActMovement^.prStroke^ * mrMinPositionFactor;
   mrMaxLimitPosition := (1.0 - rStartFactor) * mActMovement^.prPosition^ + rStartFactor * mActMovement^.prIdentPosition^;
   IF (mActMovement^.prPosition^ - mActMovement^.prIdentPosition^) > 0.0 THEN
      rMinStopRamp := rMinStrokeFactor * rRefSpeedLimit  * rRefSpeedLimit / ABS(mActMovement^.prIdentPosition^ - mActMovement^.prPosition^);
   ELSE
      rMinStopRamp := 0.0;
   END_IF;
   mActMovement^.prStopRamp^ := MAX(mActMovement^.pConstFwdVis^.Velocity.Output.rRamp, rMinStopRamp);
   mrMinLimitPosition := mActMovement^.prIdentPosition^ + 0.5 * rRefSpeedLimit  * rRefSpeedLimit / mActMovement^.prStopRamp^;
END_IF;
mActMovement^.pbMoveIdent^ := TRUE;
bMoveIdentDone := FALSE;

bMinFwdDetected := FALSE;

mrRefVelocity := rRefSpeedLimit;
mrRefPressure := rMaxRefPressureLimit;

aStartMeasurement();

bStopUnstable := FALSE;
bTimeOut := FALSE;
IF rRefSpeedLimit > 0.0 THEN
   rMoveStrokeTime := mActMovement^.prStroke^ / rRefSpeedLimit;
ELSE
   rMoveStrokeTime := 0.0;
END_IF;
dMaxMoveTime := T#5s + LINT_TO_TIME(REAL_TO_LINT(rMoveStrokeTime*1.0e6));
IF (dMaxMoveTime > dMoveTimeLimit) THEN
   dMaxMoveTime := dMoveTimeLimit;
   bMoveTimeLimited := TRUE;
   rStartPosition := mActMovement^.prPosition^;
   IF (mActMovement^.bPositionIncreasingFwd) THEN
      rMinMovementPosition := rStartPosition + 0.1 * (mrMaxLimitPosition - mrMinLimitPosition);
   ELSE;
      rMinMovementPosition := rStartPosition - 0.1 * (mrMaxLimitPosition - mrMinLimitPosition );
   END_IF;
ELSE
   bMoveTimeLimited := FALSE;
END_IF;
TimeOut(IN := FALSE,
        PT := dMaxMoveTime);
IF (mActMovement^.pdMaxMoveTimeFwd^ < dMaxMoveTime + dMoveTimeOffset) THEN
   mActMovement^.pdMaxMoveTimeFwd^ := dMaxMoveTime + dMoveTimeOffset;
END_IF;
mActMovement^.prVelocityFwd^ := rRefSpeedLimit;

sWriteSpeedLimit := REAL_TO_STRING(rRefSpeedLimit);
dummy := Print('Calib min output: act. min output: %s', sWriteSpeedLimit);
miErrorNo := cIdentSpeedMinFwdIdent;

;#END_EDIT_BLOCK END_ACTION (*ADoCalib*)
ACTION AStartMovementFwd: #BEGIN_EDIT_BLOCK
evStartRequestData.DeviceId := mActMovement^.DeviceId;
evStartRequestData.MoveDir := cMoveFwd;
IF mActMovement^.MoveId > cMoveNone THEN
   evStartRequestData.MoveId := mActMovement^.MoveId;
ELSE
   evStartRequestData.MoveId := cMoveFwd;
END_IF;
SET_EVENT(evStartRequest, evStartRequestData);

;#END_EDIT_BLOCK END_ACTION (*AStartMovementFwd*)
ACTION ACheckActMovementFwdReady: #BEGIN_EDIT_BLOCK
fbCheckReady(DeviceId := evStartRequestData.DeviceId);

TimeOut(IN := TRUE);
IF (fbCheckReady.bReady) THEN
   aStopMeasurement();
   aStopMovementFwd();
   bMoveIdentDone := TRUE;
ELSIF (TimeOut.Q) THEN
   aStopMeasurement();
   aStopMovementFwd();
   IF (bMoveTimeLimited) AND
     ((mActMovement^.bPositionIncreasingFwd AND (mActMovement^.prPosition^ > rMinMovementPosition)) OR
      (NOT mActMovement^.bPositionIncreasingFwd AND (mActMovement^.prPosition^ < rMinMovementPosition))) THEN
      bMoveIdentDone := TRUE;
      dummy := Print('Calib min output: max move time reached with act. min output %s', sWriteSpeedLimit);
   ELSE
      bTimeOut := TRUE;
      dummy := Print('Calib min output: timeout with act. min output %s', sWriteSpeedLimit);
   END_IF;
ELSIF (abSpeedMeasure.aMeasure.bSpeedUnStable) THEN
   aStopMeasurement();
   aStopMovementFwd();
   bStopUnstable := TRUE;
   dummy := Print('Calib min output: unstable speed with act. min output %s', sWriteSpeedLimit);
END_IF;

;#END_EDIT_BLOCK END_ACTION (*ACheckActMovementFwdReady*)
ACTION AStopMovementFwd: #BEGIN_EDIT_BLOCK
mActMovement^.prStopRamp^ := 0.0;
mActMovement^.pConstFwdVis^ := ConstVisFwd;
mActMovement^.pdMaxMoveTimeFwd^ := dMaxMoveTimeSaveFwd;

TimeOut(IN := FALSE);

;#END_EDIT_BLOCK END_ACTION (*AStopMovementFwd*)
STEP S_StopIdentFwd:
AStopIdentFwd (P);
END_STEP

ACTION AStopIdentFwd: #BEGIN_EDIT_BLOCK
aStopMovementFwd();
aStopMovementError(sMovementName := CONCAT(sMoveName, ' min ident Fwd'));

;#END_EDIT_BLOCK END_ACTION (*AStopIdentFwd*)
STEP S_CHECK_ALARMS_FWD:
END_STEP

STEP S_WRITE_FWD:
AWriteFwd (P);
END_STEP

ACTION AWriteFwd: #BEGIN_EDIT_BLOCK
abSpeedMeasure.aGetMaxValues(rMaxSpeed => mrMaxVelocity,
                             rMaxPressure => mrMaxPressure,
                             bPressureLimitReached => mbPressureLimitReached,
                             bSpeedLimitReached => mbVelocityLimitReached);
IF mbprActPressureLinked THEN
   rMaxPressureFwd := MAX(rMaxPressureFwd,mrMaxPressure);
   dummy := Print('Calib min output: with act. min output %s max pressure %f needed', sWriteSpeedLimit, mrMaxPressure);
END_IF;
sFileName := CONCAT(sMoveName,"_MINSPEED_FWD_");
aWriteLog(sFileName := sFileName,
          iFileCounter := iFileCounter,
          bDeleteFiles := TRUE);
iFileCounter := iFileCounter + 1;

;#END_EDIT_BLOCK END_ACTION (*AWriteFwd*)
STEP S_AbortedWriteFwd:
AStopMoveErrorWriteFwd (P);
END_STEP

ACTION AStopMoveErrorWriteFwd: #BEGIN_EDIT_BLOCK
mActMovement^.Status := tnCalibState_Error;

;#END_EDIT_BLOCK END_ACTION (*AStopMoveErrorWriteFwd*)
STEP S_CHECK_MINSPEED_FWD:
ACheckMinSpeedFwd (P);
END_STEP

ACTION ACheckMinSpeedFwd: #BEGIN_EDIT_BLOCK
aCalcMinSpeedOutput(rMaxSpeedLimit := mActMovement^.prVelocityLimitFwd^,
                    rActRefSpeed := rRefSpeedLimit,
                    rActMinSpeed := abSpeedMeasure.aGetMaxValues.rMaxSpeed,
                    bUnstable := abSpeedMeasure.aGetMaxValues.bSpeedLimitUnStable,
                    bTimeOut := bTimeOut);
bMinFwdDetected := aCalcMinSpeedOutput.bMinDetected;
IF (bMinFwdDetected) THEN
   rSpeedLimitFwd := aCalcMinSpeedOutput.rMinSpeed;
   dummy := Print('Calib min output %s Fwd finished: min output fwd = %f$N', sMoveName, rSpeedLimitFwd);
ELSE
   bMinFwdRetry := TRUE;
   rRefSpeedLimit := aCalcMinSpeedOutput.rRefSpeed;
   aCalcMinSpeedOutput.bStart := FALSE;
END_IF;

mActMovement^.pConstFwdVis^ := ConstVisFwd;
mActMovement^.prVelocityFwd^ := rSpeedLimitFwd;
mActMovement^.pdMaxMoveTimeFwd^ := dMaxMoveTimeSaveFwd;

;#END_EDIT_BLOCK END_ACTION (*ACheckMinSpeedFwd*)
STEP S_ReadyMinFwdDetected:
AReadyMinFwdDetected (N);
END_STEP

ACTION AReadyMinFwdDetected: #BEGIN_EDIT_BLOCK
fbCheckReady(DeviceId := mActMovement^.DeviceId);

;#END_EDIT_BLOCK END_ACTION (*AReadyMinFwdDetected*)
STEP S_ReadyMinFwdRetry:
AReadyMinFwdRetry (N);
END_STEP

ACTION AReadyMinFwdRetry: #BEGIN_EDIT_BLOCK
fbCheckReady(DeviceId := mActMovement^.DeviceId);

;#END_EDIT_BLOCK END_ACTION (*AReadyMinFwdRetry*)
STEP S_MinFwdRetry:
AStartMovementFwdBwd (P);
ACheckActMovementFwdBwdReady (N);
AStopMovementFwdBwd (P0);
END_STEP

ACTION AStartMovementFwdBwd: #BEGIN_EDIT_BLOCK
bMoveBwdDone := FALSE;
miErrorNo := cIdentSpeedMinFwdStart;
aStartMovementBwd();

;#END_EDIT_BLOCK END_ACTION (*AStartMovementFwdBwd*)
ACTION ACheckActMovementFwdBwdReady: #BEGIN_EDIT_BLOCK
fbCheckReady(DeviceId := evStartRequestData.DeviceId);
IF fbCheckReady.bReady THEN
   bMoveBwdDone := TRUE;
END_IF;

;#END_EDIT_BLOCK END_ACTION (*ACheckActMovementFwdBwdReady*)
ACTION AStopMovementFwdBwd: #BEGIN_EDIT_BLOCK
aStopMovementBwd();

;#END_EDIT_BLOCK END_ACTION (*AStopMovementFwdBwd*)
STEP S_StopMoveBwd:
AStopMoveErrorBwdFwd (P);
END_STEP

ACTION AStopMoveErrorBwdFwd: #BEGIN_EDIT_BLOCK
aStopMovementError(sMovementName := CONCAT(sMoveName, ' min ident Fwd: Bwd to start position'));

;#END_EDIT_BLOCK END_ACTION (*AStopMoveErrorBwdFwd*)
STEP S_CHECK_ALARMS_RETRYFWD:
END_STEP

STEP S_InitStartMovementBwdFwd:
AInitStartMovementBwdFwd (P);
ACheckInitMovementBwdFwdReady (N);
AStopInitMovementBwdFwd (P0);
END_STEP

ACTION AInitStartMovementBwdFwd: #BEGIN_EDIT_BLOCK
bMoveFwdDone := FALSE;
miErrorNo := cIdentSpeedMinFwdInit;
aStartMovementFwd();

;#END_EDIT_BLOCK END_ACTION (*AInitStartMovementBwdFwd*)
ACTION ACheckInitMovementBwdFwdReady: #BEGIN_EDIT_BLOCK
fbCheckReady(DeviceId := evStartRequestData.DeviceId);
IF fbCheckReady.bReady THEN
   bMoveFwdDone := TRUE;
END_IF;

;#END_EDIT_BLOCK END_ACTION (*ACheckInitMovementBwdFwdReady*)
ACTION AStopInitMovementBwdFwd: #BEGIN_EDIT_BLOCK
aStopMovementFwd();

;#END_EDIT_BLOCK END_ACTION (*AStopInitMovementBwdFwd*)
STEP S_StopInitMoveFwd:
AStopMoveErrorInitFwd (P);
END_STEP

ACTION AStopMoveErrorInitFwd: #BEGIN_EDIT_BLOCK
aStopMovementError(sMovementName := CONCAT(sMoveName, ' min ident Bwd: Fwd to initial position'));

;#END_EDIT_BLOCK END_ACTION (*AStopMoveErrorInitFwd*)
STEP S_CHECK_ALARMS_STARTBWD:
END_STEP

STEP S_INITCALIB_BWD:
AInitCalibBwd (P);
END_STEP

ACTION AInitCalibBwd: #BEGIN_EDIT_BLOCK
iFileCounter := 1;
IF (CHECK_REF(mActMovement^.prSizeFactorBwd^)) THEN
   IF (mActMovement^.prSizeFactorBwd^ > 0.0) THEN
      rVelocitSizeFactor := mActMovement^.prSizeFactorBwd^;
   END_IF;
ELSE
   rVelocitSizeFactor := 1.0;
END_IF;
rRefSpeedLimit := 0.01 * mActMovement^.prVelocityLimitBwd^;
rMaxPressureLimit := mActMovement^.prMaxPressureBwd^;
IF CHECK_REF(mActMovement^.prMaxPressureBwdHydr^) THEN
   rMaxRefPressureLimit := mActMovement^.prMaxPressureBwdHydr^;
   IF (rMaxRefPressureLimit > 0.0) THEN
      rPressureFactorBwd := rMaxPressureLimit / rMaxRefPressureLimit;
   ELSE
      rPressureFactorBwd := 1.0;
   END_IF;
ELSE
   rMaxRefPressureLimit := mActMovement^.prMaxPressureFwd^;
   rPressureFactorBwd := 1.0;
END_IF;

aCalcMinSpeedOutput.bStart := TRUE;

dummy := Print('Calib min output %s Bwd started', sMoveName);

;#END_EDIT_BLOCK END_ACTION (*AInitCalibBwd*)
STEP S_CALIB_BWD:
ADoCalibBwd (P);
AStartMovementBwd (P);
ACheckActMovementBwdReady (N);
AStopMovementBwd (P0);
END_STEP

ACTION ADoCalibBwd: #BEGIN_EDIT_BLOCK
mActMovement^.pConstBwdVis^.Velocity.Output.rOutputValue := rRefSpeedLimit * rVelocitSizeFactor;
mActMovement^.pConstBwdVis^.Velocity.rMinOutput := 0.0;
mActMovement^.pConstBwdVis^.Pressure.Output.rOutputValue := MAX(mActMovement^.pConstBwdVis^.Pressure.Output.rOutputValue, rMaxPressureLimit);
mActMovement^.pConstBwdVis^.Pressure.Output.rRamp := MAX(1.0e10, ConstVisBwd.Pressure.Output.rRamp);
IF mActMovement^.bPositionIncreasingFwd THEN
   mActMovement^.prIdentPosition^ := mActMovement^.prStroke^ * mrMinPositionFactor;
   mrMaxLimitPosition := rStartFactor * mActMovement^.prIdentPosition^ + (1.0 - rStartFactor) * mActMovement^.prPosition^;
   IF (mActMovement^.prPosition^ - mActMovement^.prIdentPosition^) > 0.0 THEN
      rMinStopRamp := rMinStrokeFactor * rRefSpeedLimit  * rRefSpeedLimit / ABS(mActMovement^.prIdentPosition^ - mActMovement^.prPosition^);
   ELSE
      rMinStopRamp := 0.0;
   END_IF;
   mActMovement^.prStopRamp^ := MAX(mActMovement^.pConstBwdVis^.Velocity.Output.rRamp, rMinStopRamp);
   mrMinLimitPosition := mActMovement^.prIdentPosition^ + 0.5 * rRefSpeedLimit  * rRefSpeedLimit / mActMovement^.prStopRamp^;
ELSE
   mActMovement^.prIdentPosition^ := mActMovement^.prStroke^ * mrMaxPositionFactor;
   mrMinLimitPosition := rStartFactor * mActMovement^.prPosition^ + (1.0 - rStartFactor) * mActMovement^.prIdentPosition^;
   IF (mActMovement^.prIdentPosition^ - mActMovement^.prPosition^) > 0.0 THEN
      rMinStopRamp := rMinStrokeFactor * rRefSpeedLimit  * rRefSpeedLimit / ABS(mActMovement^.prIdentPosition^ - mActMovement^.prPosition^);
   ELSE
      rMinStopRamp := 0.0;
   END_IF;
   mActMovement^.prStopRamp^ := MAX(mActMovement^.pConstBwdVis^.Velocity.Output.rRamp, rMinStopRamp);
   mrMaxLimitPosition := mActMovement^.prIdentPosition^ - 0.5 * rRefSpeedLimit  * rRefSpeedLimit / mActMovement^.prStopRamp^;
END_IF;
mActMovement^.pbMoveIdent^ := TRUE;

bMoveIdentDone := FALSE;

mrRefVelocity := rRefSpeedLimit;
mrRefPressure := rMaxRefPressureLimit;

aStartMeasurement();

bStopUnstable := FALSE;
bTimeOut := FALSE;
IF rRefSpeedLimit > 0.0 THEN
   rMoveStrokeTime := mActMovement^.prStroke^ / rRefSpeedLimit;
ELSE
   rMoveStrokeTime := 0.0;
END_IF;
dMaxMoveTime := T#5s + LINT_TO_TIME(REAL_TO_LINT(rMoveStrokeTime*1.0e6));
IF (dMaxMoveTime > dMoveTimeLimit) THEN
   dMaxMoveTime := dMoveTimeLimit;
   bMoveTimeLimited := TRUE;
   rStartPosition := mActMovement^.prPosition^;
   IF (mActMovement^.bPositionIncreasingFwd) THEN
      rMinMovementPosition := rStartPosition - 0.1 * (mrMaxLimitPosition - mrMinLimitPosition);
   ELSE;
      rMinMovementPosition := rStartPosition + 0.1 * (mrMaxLimitPosition - mrMinLimitPosition );
   END_IF;
ELSE
   bMoveTimeLimited := FALSE;
END_IF;

TimeOut(IN := FALSE,
        PT := dMaxMoveTime);
IF (mActMovement^.pdMaxMoveTimeBwd^ < dMaxMoveTime + dMoveTimeOffset) THEN
   mActMovement^.pdMaxMoveTimeBwd^ := dMaxMoveTime + dMoveTimeOffset;
END_IF;
mActMovement^.prVelocityBwd^ := rRefSpeedLimit;

sWriteSpeedLimit := REAL_TO_STRING(rRefSpeedLimit);
dummy := Print('Calib min output: act. min output: %s', sWriteSpeedLimit);
miErrorNo := cIdentSpeedMinBwdIdent;

;#END_EDIT_BLOCK END_ACTION (*ADoCalibBwd*)
ACTION AStartMovementBwd: #BEGIN_EDIT_BLOCK
evStartRequestData.DeviceId := mActMovement^.DeviceId;
evStartRequestData.MoveDir := cMoveBwd;
IF mActMovement^.MoveId > cMoveNone THEN
   evStartRequestData.MoveId := cMoveDecompAftPlast;
ELSE
   evStartRequestData.MoveId := cMoveBwd;
END_IF;
SET_EVENT(evStartRequest, evStartRequestData);

;#END_EDIT_BLOCK END_ACTION (*AStartMovementBwd*)
ACTION ACheckActMovementBwdReady: #BEGIN_EDIT_BLOCK
fbCheckReady(DeviceId := evStartRequestData.DeviceId);

TimeOut(IN :=TRUE);
IF fbCheckReady.bReady THEN
   aStopMeasurement();
   aStopMovementBwd();
   bMoveIdentDone := TRUE;
ELSIF TimeOut.Q THEN
   aStopMeasurement();
   aStopMovementBwd();
   IF (bMoveTimeLimited) AND
     ((mActMovement^.bPositionIncreasingFwd AND (mActMovement^.prPosition^ < rMinMovementPosition)) OR
      (NOT mActMovement^.bPositionIncreasingFwd AND (mActMovement^.prPosition^ > rMinMovementPosition))) THEN
      bMoveIdentDone := TRUE;
      dummy := Print('Calib min output: max move time reached with act. min output %s', sWriteSpeedLimit);
   ELSE
      bTimeOut := TRUE;
      dummy := Print('Calib min output: timeout with act. min output %s', sWriteSpeedLimit);
   END_IF;
ELSIF (abSpeedMeasure.aMeasure.bSpeedUnStable) THEN
   aStopMeasurement();
   aStopMovementBwd();
   bStopUnstable := TRUE;
   sWriteSpeedLimit := REAL_TO_STRING(rRefSpeedLimit);
   dummy := Print('Calib min output: unstable speed with act. min output %s', sWriteSpeedLimit);
END_IF;

;#END_EDIT_BLOCK END_ACTION (*ACheckActMovementBwdReady*)
ACTION AStopMovementBwd: #BEGIN_EDIT_BLOCK
mActMovement^.pConstBwdVis^ := ConstVisBwd;
mActMovement^.pdMaxMoveTimeBwd^ := dMaxMoveTimeSaveBwd;

TimeOut(IN := FALSE);

;#END_EDIT_BLOCK END_ACTION (*AStopMovementBwd*)
STEP S_StopCalibBwd:
AStopMoveErrorCalibBwd (P);
END_STEP

ACTION AStopMoveErrorCalibBwd: #BEGIN_EDIT_BLOCK
aStopMovementBwd();
aStopMovementError(sMovementName := CONCAT(sMoveName, ' min ident Bwd'));

;#END_EDIT_BLOCK END_ACTION (*AStopMoveErrorCalibBwd*)
STEP S_CHECK_ALARMS_BWD:
END_STEP

STEP S_WRITE_BWD:
AWriteBwd (P);
END_STEP

ACTION AWriteBwd: #BEGIN_EDIT_BLOCK
abSpeedMeasure.aGetMaxValues(rMaxSpeed => mrMaxVelocity,
                             rMaxPressure => mrMaxPressure,
                             bPressureLimitReached => mbPressureLimitReached,
                             bSpeedLimitReached => mbVelocityLimitReached);
IF mbprActPressureLinked THEN
   rMaxPressureBwd := MAX(rMaxPressureBwd, mrMaxPressure);
   dummy := Print('Calib min output: with act. min output %s max pressure %f needed', sWriteSpeedLimit, mrMaxPressure);
END_IF;
sFileName := CONCAT(sMoveName,"_MINSPEED_BWD_");
aWriteLog(sFileName := sFileName,
          iFileCounter := iFileCounter,
          bDeleteFiles := TRUE);
iFileCounter := iFileCounter + 1;

;#END_EDIT_BLOCK END_ACTION (*AWriteBwd*)
STEP S_CHECK_MINSPEED_BWD:
ACheckMinSpeedBwd (P);
END_STEP

ACTION ACheckMinSpeedBwd: #BEGIN_EDIT_BLOCK
aCalcMinSpeedOutput(rMaxSpeedLimit := mActMovement^.prVelocityLimitBwd^,
                    rActRefSpeed := rRefSpeedLimit,
                    rActMinSpeed := abSpeedMeasure.aGetMaxValues.rMaxSpeed,
                    bUnstable := abSpeedMeasure.aGetMaxValues.bSpeedLimitUnStable,
                    bTimeOut := bTimeOut);
bMinBwdDetected := aCalcMinSpeedOutput.bMinDetected;
IF (bMinBwdDetected) THEN
   rSpeedLimitBwd := aCalcMinSpeedOutput.rMinSpeed;
   dummy := Print('Calib min output %s Bwd finished: min output bwd = %f$N', sMoveName, rSpeedLimitBwd);
ELSE
   bMinBwdRetry := TRUE;
   rRefSpeedLimit := aCalcMinSpeedOutput.rRefSpeed;
   aCalcMinSpeedOutput.bStart := FALSE;
END_IF;

mActMovement^.pConstBwdVis^ := ConstVisBwd;
mActMovement^.prVelocityBwd^ := rSpeedLimitBwd;
mActMovement^.pdMaxMoveTimeBwd^ := dMaxMoveTimeSaveBwd;

;#END_EDIT_BLOCK END_ACTION (*ACheckMinSpeedBwd*)
STEP S_ReadyMinBwdRetry:
AReadyMinBwdRetry (N);
END_STEP

ACTION AReadyMinBwdRetry: #BEGIN_EDIT_BLOCK
fbCheckReady(DeviceId := mActMovement^.DeviceId);

;#END_EDIT_BLOCK END_ACTION (*AReadyMinBwdRetry*)
STEP S_MinBwdRetry:
AStartMovementBwdFwd (P);
ACheckActMovementBwdFwdReady (N);
AStopMovementBwdFwd (P0);
END_STEP

ACTION AStartMovementBwdFwd: #BEGIN_EDIT_BLOCK
bMoveFwdDone := FALSE;
miErrorNo := cIdentSpeedMinBwdStart;
aStartMovementFwd();

;#END_EDIT_BLOCK END_ACTION (*AStartMovementBwdFwd*)
ACTION ACheckActMovementBwdFwdReady: #BEGIN_EDIT_BLOCK
fbCheckReady(DeviceId := evStartRequestData.DeviceId);
IF fbCheckReady.bReady THEN
   bMoveFwdDone := TRUE;
END_IF;

;#END_EDIT_BLOCK END_ACTION (*ACheckActMovementBwdFwdReady*)
ACTION AStopMovementBwdFwd: #BEGIN_EDIT_BLOCK
aStopMovementFwd();

;#END_EDIT_BLOCK END_ACTION (*AStopMovementBwdFwd*)
STEP S_StopMoveFwd:
AStopMoveErrorFwd (P);
END_STEP

ACTION AStopMoveErrorFwd: #BEGIN_EDIT_BLOCK
aStopMovementError(sMovementName := CONCAT(sMoveName, ' min ident Bwd: Fwd to start position'));

;#END_EDIT_BLOCK END_ACTION (*AStopMoveErrorFwd*)
STEP S_CHECK_ALARMS_RETRYBWD:
END_STEP

STEP S_MoveEndBwd:
AMoveEndBwd (P);
ACheckMoveEndBwdReady (N);
AMoveEndBwdReady (P0);
END_STEP

ACTION AMoveEndBwd: #BEGIN_EDIT_BLOCK
bMoveBwdDone := FALSE;

IF mActMovement^.bPositionIncreasingFwd THEN
   mActMovement^.prIdentPosition^ := mrBwdStopPosition;
ELSE
   mActMovement^.prIdentPosition^ := mActMovement^.prStroke^ - mrBwdStopPosition;
END_IF;
mActMovement^.prStopRamp^ := 1.0e10;
mActMovement^.pConstBwdVis^.Pressure.Output.rRamp := MAX(1.0e20,mActMovement^.pConstBwdVis^.Pressure.Output.rRamp);
mActMovement^.pConstBwdVis^.Pressure.rMinOutput := 0.1 * rMaxPressureLimit;
mActMovement^.pbMoveIdent^ := TRUE;

evStartRequestData.DeviceId := mActMovement^.DeviceId;
evStartRequestData.MoveDir := cMoveBwd;
IF mActMovement^.MoveId > cMoveNone THEN
   evStartRequestData.MoveId := cMoveDecompAftPlast;
ELSE
   evStartRequestData.MoveId := cMoveBwd;
END_IF;
miErrorNo := cIdentSpeedMinEnd;
SET_EVENT(evStartRequest, evStartRequestData);

;#END_EDIT_BLOCK END_ACTION (*AMoveEndBwd*)
ACTION ACheckMoveEndBwdReady: #BEGIN_EDIT_BLOCK
fbCheckReady(DeviceId := evStartRequestData.DeviceId);
IF fbCheckReady.bReady THEN
   bMoveBwdDone := TRUE;
END_IF;

;#END_EDIT_BLOCK END_ACTION (*ACheckMoveEndBwdReady*)
ACTION AMoveEndBwdReady: #BEGIN_EDIT_BLOCK
aStopMovementBwd();

;#END_EDIT_BLOCK END_ACTION (*AMoveEndBwdReady*)
STEP S_StopMoveEndBwd:
AStopMoveErrorEndBwd (P);
END_STEP

ACTION AStopMoveErrorEndBwd: #BEGIN_EDIT_BLOCK
aStopMovementError(sMovementName := CONCAT(sMoveName, ' min ident: Bwd to end position'));

;#END_EDIT_BLOCK END_ACTION (*AStopMoveErrorEndBwd*)
STEP S_Done:
ADone (P);
END_STEP

ACTION ADone: #BEGIN_EDIT_BLOCK
mActMovement^.Status := tnCalibState_Done;
sv_GlobalIdentMinSpeedStatus.Status := tnCalibState_Done;

mActMovement^.prVelocityFwd^ := rSpeedLimitFwd;
mActMovement^.prVelocityBwd^ := rSpeedLimitBwd;
IF mbprActPressureLinked THEN
   IF CHECK_REF(mActMovement^.prIdentPressureFwd^) THEN
      aRound(rActNumber := rMaxPressureFwd, rStep := rPressureStep);
      mActMovement^.prIdentPressureFwd^ := MAX(mActMovement^.prIdentPressureFwd^, aRound.rRoundedNumber * rPressureFactorFwd);
   END_IF;
   IF CHECK_REF(mActMovement^.prIdentPressureBwd^) THEN
      aRound(rActNumber := rMaxPressureBwd, rStep := rPressureStep);
      mActMovement^.prIdentPressureBwd^ := MAX(mActMovement^.prIdentPressureBwd^, aRound.rRoundedNumber * rPressureFactorBwd);
   END_IF;
END_IF;

;#END_EDIT_BLOCK END_ACTION (*ADone*)

(* transitions *)
TRANSITION Trans47 (* Trans47 *) FROM S_RESET TO S_STOP :=  #BEGIN_EDIT_BLOCK
mbLogFileSaved
;#END_EDIT_BLOCK
END_TRANSITION

TRANSITION TRestart (* TRestart *) FROM S_STOP TO S_INIT :=  #BEGIN_EDIT_BLOCK
TRUE
;#END_EDIT_BLOCK
END_TRANSITION

TRANSITION TMoveStartBwd (* TMoveStartBwd *) FROM S_INIT TO S_MoveStartBwd :=  #BEGIN_EDIT_BLOCK
TRUE

;#END_EDIT_BLOCK
END_TRANSITION

TRANSITION TInitBwd (* TInitBwd *) FROM S_MoveStartBwd TO S_CHECK_ALARMS_INITBWD :=  #BEGIN_EDIT_BLOCK
bMoveBwdDone
;#END_EDIT_BLOCK
END_TRANSITION

GO_ON_TRANSITION TStopMoveStartBwd (* TStopMoveStartBwd *) FROM S_MoveStartBwd TO S_StopMoveStartBwd :=  #BEGIN_EDIT_BLOCK
sv_GlobalIdentMinSpeedStatus.Status = tnCalibState_Aborted OR
sv_GlobalIdentMinSpeedStatus.Status = tnCalibState_None
OR sv_iPendingAlarms <> 0
OR mActMovement^.bRedo = FALSE
;#END_EDIT_BLOCK
END_TRANSITION

GO_ON_TRANSITION TReset (* TReset *) FROM S_StopMoveStartBwd TO S_RESET :=  #BEGIN_EDIT_BLOCK
TRUE
;#END_EDIT_BLOCK
END_TRANSITION

TRANSITION TStartIdent (* TStartIdent *) FROM S_CHECK_ALARMS_INITBWD TO S_INITCALIB_FWD :=  #BEGIN_EDIT_BLOCK
S_CHECK_ALARMS_INITBWD.T > T#100ms
;#END_EDIT_BLOCK
END_TRANSITION

GO_ON_TRANSITION TStopInitBwd (* TStopInitBwd *) FROM S_CHECK_ALARMS_INITBWD TO S_StopMoveStartBwd :=  #BEGIN_EDIT_BLOCK
sv_iPendingAlarms <> 0
;#END_EDIT_BLOCK
END_TRANSITION

TRANSITION TDelay1 (* TDelay1 *) FROM S_INITCALIB_FWD TO S_CALIB_FWD :=  #BEGIN_EDIT_BLOCK
S_INITCALIB_FWD.T>T#100ms
;#END_EDIT_BLOCK
END_TRANSITION

TRANSITION TMoveIdentFwdDone (* TMoveIdentFwdDone *) FROM S_CALIB_FWD TO S_CHECK_ALARMS_FWD :=  #BEGIN_EDIT_BLOCK
bMoveIdentDone OR
bTimeOut OR
bStopUnstable
;#END_EDIT_BLOCK
END_TRANSITION

GO_ON_TRANSITION TStopIdentFwd (* TStopIdentFwd *) FROM S_CALIB_FWD TO S_StopIdentFwd :=  #BEGIN_EDIT_BLOCK
sv_GlobalIdentMinSpeedStatus.Status = tnCalibState_Aborted OR
sv_GlobalIdentMinSpeedStatus.Status = tnCalibState_None
OR sv_iPendingAlarms <> 0
OR mActMovement^.bRedo = FALSE
;#END_EDIT_BLOCK
END_TRANSITION

GO_ON_TRANSITION TReset1 (* TReset1 *) FROM S_StopIdentFwd TO S_RESET :=  #BEGIN_EDIT_BLOCK
TRUE
;#END_EDIT_BLOCK
END_TRANSITION

TRANSITION TStartWriteFwd (* TStartWriteFwd *) FROM S_CHECK_ALARMS_FWD TO S_WRITE_FWD :=  #BEGIN_EDIT_BLOCK
S_CHECK_ALARMS_FWD.T > T#100ms
;#END_EDIT_BLOCK
END_TRANSITION

GO_ON_TRANSITION TStopIdentFwd2 (* TStopIdentFwd2 *) FROM S_CHECK_ALARMS_FWD TO S_StopIdentFwd :=  #BEGIN_EDIT_BLOCK
sv_iPendingAlarms <> 0
;#END_EDIT_BLOCK
END_TRANSITION

TRANSITION TWriteFwd (* TWriteFwd *) FROM S_WRITE_FWD TO S_CHECK_MINSPEED_FWD :=  #BEGIN_EDIT_BLOCK
mbLogFileSaved
;#END_EDIT_BLOCK
END_TRANSITION

GO_ON_TRANSITION TAbortedWriteFwd (* TAbortedWriteFwd *) FROM S_WRITE_FWD TO S_AbortedWriteFwd :=  #BEGIN_EDIT_BLOCK
sv_GlobalIdentMinSpeedStatus.Status = tnCalibState_Aborted
;#END_EDIT_BLOCK
END_TRANSITION

GO_ON_TRANSITION TResetAbortedWriteFwd (* TResetAbortedWriteFwd *) FROM S_AbortedWriteFwd TO S_RESET :=  #BEGIN_EDIT_BLOCK
TRUE
;#END_EDIT_BLOCK
END_TRANSITION

TRANSITION TMinFwdDetected (* TMinFwdDetected *) FROM S_CHECK_MINSPEED_FWD TO S_ReadyMinFwdDetected :=  #BEGIN_EDIT_BLOCK
bMinFwdDetected
;#END_EDIT_BLOCK
END_TRANSITION

TRANSITION TReadyMinFwdDetected (* Trans49 *) FROM S_ReadyMinFwdDetected TO S_InitStartMovementBwdFwd :=  #BEGIN_EDIT_BLOCK
fbCheckReady.bReady
;#END_EDIT_BLOCK
END_TRANSITION

TRANSITION Trans15 (* Trans15 *) FROM S_CHECK_MINSPEED_FWD TO S_ReadyMinFwdRetry :=  #BEGIN_EDIT_BLOCK
bMinFwdRetry
;#END_EDIT_BLOCK
END_TRANSITION

TRANSITION TReadyMinFwdRetry (* Trans49 *) FROM S_ReadyMinFwdRetry TO S_MinFwdRetry :=  #BEGIN_EDIT_BLOCK
fbCheckReady.bReady
;#END_EDIT_BLOCK
END_TRANSITION

TRANSITION TMoveBwdDone (* TMoveBwdDone *) FROM S_MinFwdRetry TO S_CHECK_ALARMS_RETRYFWD :=  #BEGIN_EDIT_BLOCK
bMoveBwdDone
;#END_EDIT_BLOCK
END_TRANSITION

GO_ON_TRANSITION TStopMoveBwd (* TStopMoveBwd *) FROM S_MinFwdRetry TO S_StopMoveBwd :=  #BEGIN_EDIT_BLOCK
sv_GlobalIdentMinSpeedStatus.Status = tnCalibState_Aborted OR
sv_GlobalIdentMinSpeedStatus.Status = tnCalibState_None
OR sv_iPendingAlarms <> 0
OR mActMovement^.bRedo = FALSE

;#END_EDIT_BLOCK
END_TRANSITION

TRANSITION TReset2 (* TReset2 *) FROM S_StopMoveBwd TO S_RESET :=  #BEGIN_EDIT_BLOCK
TRUE
;#END_EDIT_BLOCK
END_TRANSITION

TRANSITION TRetryFwd (* TRetryFwd *) FROM S_CHECK_ALARMS_RETRYFWD TO S_CALIB_FWD :=  #BEGIN_EDIT_BLOCK
S_CHECK_ALARMS_RETRYFWD.T > T#1s
;#END_EDIT_BLOCK
END_TRANSITION

GO_ON_TRANSITION TStopIdentFwd4 (* TStopIdentFwd4 *) FROM S_CHECK_ALARMS_RETRYFWD TO S_StopMoveBwd :=  #BEGIN_EDIT_BLOCK
sv_iPendingAlarms <> 0
;#END_EDIT_BLOCK
END_TRANSITION

TRANSITION Trans35 (* Trans35 *) FROM S_InitStartMovementBwdFwd TO S_CHECK_ALARMS_STARTBWD :=  #BEGIN_EDIT_BLOCK
bMoveFwdDone
;#END_EDIT_BLOCK
END_TRANSITION

GO_ON_TRANSITION TStopInitMoveFwd (* TStopInitMoveFwd *) FROM S_InitStartMovementBwdFwd TO S_StopInitMoveFwd :=  #BEGIN_EDIT_BLOCK
sv_GlobalIdentMinSpeedStatus.Status = tnCalibState_Aborted OR
sv_GlobalIdentMinSpeedStatus.Status = tnCalibState_None
OR sv_iPendingAlarms <> 0
OR mActMovement^.bRedo = FALSE
;#END_EDIT_BLOCK
END_TRANSITION

TRANSITION TResetInitMoveFwd (* TResetInitMoveFwd *) FROM S_StopInitMoveFwd TO S_RESET :=  #BEGIN_EDIT_BLOCK
TRUE
;#END_EDIT_BLOCK
END_TRANSITION

TRANSITION TStartInitBwd (* TStartInitBwd *) FROM S_CHECK_ALARMS_STARTBWD TO S_INITCALIB_BWD :=  #BEGIN_EDIT_BLOCK
S_CHECK_ALARMS_STARTBWD.T > T#100ms
;#END_EDIT_BLOCK
END_TRANSITION

GO_ON_TRANSITION TStopIdentFwd3 (* TStopIdentFwd3 *) FROM S_CHECK_ALARMS_STARTBWD TO S_StopInitMoveFwd :=  #BEGIN_EDIT_BLOCK
sv_iPendingAlarms <> 0
;#END_EDIT_BLOCK
END_TRANSITION

TRANSITION TInitCalibBwd (* TInitCalibBwd *) FROM S_INITCALIB_BWD TO S_CALIB_BWD :=  #BEGIN_EDIT_BLOCK
S_INITCALIB_BWD.T>T#1s
;#END_EDIT_BLOCK
END_TRANSITION

TRANSITION Trans14 (* Trans14 *) FROM S_CALIB_BWD TO S_CHECK_ALARMS_BWD :=  #BEGIN_EDIT_BLOCK
bMoveIdentDone OR
bTimeOut OR
bStopUnstable
;#END_EDIT_BLOCK
END_TRANSITION

GO_ON_TRANSITION TStopCalibBwd (* TStopCalibBwd *) FROM S_CALIB_BWD TO S_StopCalibBwd :=  #BEGIN_EDIT_BLOCK
sv_GlobalIdentMinSpeedStatus.Status = tnCalibState_Aborted OR
sv_GlobalIdentMinSpeedStatus.Status = tnCalibState_None
OR sv_iPendingAlarms <> 0
OR mActMovement^.bRedo = FALSE
;#END_EDIT_BLOCK
END_TRANSITION
